boPin193Fault.AppScalingDivisor :=1;
boPin193Fault.AppScalingMultiplier :=1;
boPin193Fault.AppScalingOffset :=0;
boPin193Fault.AppUnit :="";
boPin193Fault.CanDefault :=0;
boPin193Fault.CanInit :=0;
boPin193Fault.CanMax :=1;
boPin193Fault.CanMin :=0;
boPin193Fault.CanUnit :="";
boPin193Fault.Description :="for the Neotec diag pages";
boPin193Fault.ErrorReaction := eErrorReaction.ERSIG_DFLT;
boPin193Fault.ReceiverAdress :=1;
boPin193Fault.ToolScalingDivisor :=1;
boPin193Fault.ToolScalingMultiplier :=1;
boPin193Fault.ToolScalingOffset :=0;
boPin193Fault.ToolUnit :="";

boPin169Fault.AppScalingDivisor :=1;
boPin169Fault.AppScalingMultiplier :=1;
boPin169Fault.AppScalingOffset :=0;
boPin169Fault.AppUnit :="";
boPin169Fault.CanDefault :=0;
boPin169Fault.CanInit :=0;
boPin169Fault.CanMax :=1;
boPin169Fault.CanMin :=0;
boPin169Fault.CanUnit :="";
boPin169Fault.Description :="for the Neotec diag pages";
boPin169Fault.ErrorReaction := eErrorReaction.ERSIG_DFLT;
boPin169Fault.ReceiverAdress :=1;
boPin169Fault.ToolScalingDivisor :=1;
boPin169Fault.ToolScalingMultiplier :=1;
boPin169Fault.ToolScalingOffset :=0;
boPin169Fault.ToolUnit :="";

boPin196Fault.AppScalingDivisor :=1;
boPin196Fault.AppScalingMultiplier :=1;
boPin196Fault.AppScalingOffset :=0;
boPin196Fault.AppUnit :="";
boPin196Fault.CanDefault :=0;
boPin196Fault.CanInit :=0;
boPin196Fault.CanMax :=1;
boPin196Fault.CanMin :=0;
boPin196Fault.CanUnit :="";
boPin196Fault.Description :="for the Neotec diag pages";
boPin196Fault.ErrorReaction := eErrorReaction.ERSIG_DFLT;
boPin196Fault.ReceiverAdress :=1;
boPin196Fault.ToolScalingDivisor :=1;
boPin196Fault.ToolScalingMultiplier :=1;
boPin196Fault.ToolScalingOffset :=0;
boPin196Fault.ToolUnit :="";

boPin172Fault.AppScalingDivisor :=1;
boPin172Fault.AppScalingMultiplier :=1;
boPin172Fault.AppScalingOffset :=0;
boPin172Fault.AppUnit :="";
boPin172Fault.CanDefault :=0;
boPin172Fault.CanInit :=0;
boPin172Fault.CanMax :=1;
boPin172Fault.CanMin :=0;
boPin172Fault.CanUnit :="";
boPin172Fault.Description :="for the Neotec diag pages";
boPin172Fault.ErrorReaction := eErrorReaction.ERSIG_DFLT;
boPin172Fault.ReceiverAdress :=1;
boPin172Fault.ToolScalingDivisor :=1;
boPin172Fault.ToolScalingMultiplier :=1;
boPin172Fault.ToolScalingOffset :=0;
boPin172Fault.ToolUnit :="";

boPin101Fault.AppScalingDivisor :=1;
boPin101Fault.AppScalingMultiplier :=1;
boPin101Fault.AppScalingOffset :=0;
boPin101Fault.AppUnit :="";
boPin101Fault.CanDefault :=0;
boPin101Fault.CanInit :=0;
boPin101Fault.CanMax :=1;
boPin101Fault.CanMin :=0;
boPin101Fault.CanUnit :="";
boPin101Fault.Description :="for the Neotec diag pages";
boPin101Fault.ErrorReaction := eErrorReaction.ERSIG_DFLT;
boPin101Fault.ReceiverAdress :=1;
boPin101Fault.ToolScalingDivisor :=1;
boPin101Fault.ToolScalingMultiplier :=1;
boPin101Fault.ToolScalingOffset :=0;
boPin101Fault.ToolUnit :="";

boPin125Fault.AppScalingDivisor :=1;
boPin125Fault.AppScalingMultiplier :=1;
boPin125Fault.AppScalingOffset :=0;
boPin125Fault.AppUnit :="";
boPin125Fault.CanDefault :=0;
boPin125Fault.CanInit :=0;
boPin125Fault.CanMax :=1;
boPin125Fault.CanMin :=0;
boPin125Fault.CanUnit :="";
boPin125Fault.Description :="for the Neotec diag pages";
boPin125Fault.ErrorReaction := eErrorReaction.ERSIG_DFLT;
boPin125Fault.ReceiverAdress :=1;
boPin125Fault.ToolScalingDivisor :=1;
boPin125Fault.ToolScalingMultiplier :=1;
boPin125Fault.ToolScalingOffset :=0;
boPin125Fault.ToolUnit :="";

boPin150Fault.AppScalingDivisor :=1;
boPin150Fault.AppScalingMultiplier :=1;
boPin150Fault.AppScalingOffset :=0;
boPin150Fault.AppUnit :="";
boPin150Fault.CanDefault :=0;
boPin150Fault.CanInit :=0;
boPin150Fault.CanMax :=1;
boPin150Fault.CanMin :=0;
boPin150Fault.CanUnit :="";
boPin150Fault.Description :="for the Neotec diag pages";
boPin150Fault.ErrorReaction := eErrorReaction.ERSIG_DFLT;
boPin150Fault.ReceiverAdress :=1;
boPin150Fault.ToolScalingDivisor :=1;
boPin150Fault.ToolScalingMultiplier :=1;
boPin150Fault.ToolScalingOffset :=0;
boPin150Fault.ToolUnit :="";

boPin174Fault.AppScalingDivisor :=1;
boPin174Fault.AppScalingMultiplier :=1;
boPin174Fault.AppScalingOffset :=0;
boPin174Fault.AppUnit :="";
boPin174Fault.CanDefault :=0;
boPin174Fault.CanInit :=0;
boPin174Fault.CanMax :=1;
boPin174Fault.CanMin :=0;
boPin174Fault.CanUnit :="";
boPin174Fault.Description :="for the Neotec diag pages";
boPin174Fault.ErrorReaction := eErrorReaction.ERSIG_DFLT;
boPin174Fault.ReceiverAdress :=1;
boPin174Fault.ToolScalingDivisor :=1;
boPin174Fault.ToolScalingMultiplier :=1;
boPin174Fault.ToolScalingOffset :=0;
boPin174Fault.ToolUnit :="";

boPin102Fault.AppScalingDivisor :=1;
boPin102Fault.AppScalingMultiplier :=1;
boPin102Fault.AppScalingOffset :=0;
boPin102Fault.AppUnit :="";
boPin102Fault.CanDefault :=0;
boPin102Fault.CanInit :=0;
boPin102Fault.CanMax :=1;
boPin102Fault.CanMin :=0;
boPin102Fault.CanUnit :="";
boPin102Fault.Description :="for the Neotec diag pages";
boPin102Fault.ErrorReaction := eErrorReaction.ERSIG_DFLT;
boPin102Fault.ReceiverAdress :=1;
boPin102Fault.ToolScalingDivisor :=1;
boPin102Fault.ToolScalingMultiplier :=1;
boPin102Fault.ToolScalingOffset :=0;
boPin102Fault.ToolUnit :="";

boPin126Fault.AppScalingDivisor :=1;
boPin126Fault.AppScalingMultiplier :=1;
boPin126Fault.AppScalingOffset :=0;
boPin126Fault.AppUnit :="";
boPin126Fault.CanDefault :=0;
boPin126Fault.CanInit :=0;
boPin126Fault.CanMax :=1;
boPin126Fault.CanMin :=0;
boPin126Fault.CanUnit :="";
boPin126Fault.Description :="for the Neotec diag pages";
boPin126Fault.ErrorReaction := eErrorReaction.ERSIG_DFLT;
boPin126Fault.ReceiverAdress :=1;
boPin126Fault.ToolScalingDivisor :=1;
boPin126Fault.ToolScalingMultiplier :=1;
boPin126Fault.ToolScalingOffset :=0;
boPin126Fault.ToolUnit :="";

boPin151Fault.AppScalingDivisor :=1;
boPin151Fault.AppScalingMultiplier :=1;
boPin151Fault.AppScalingOffset :=0;
boPin151Fault.AppUnit :="";
boPin151Fault.CanDefault :=0;
boPin151Fault.CanInit :=0;
boPin151Fault.CanMax :=1;
boPin151Fault.CanMin :=0;
boPin151Fault.CanUnit :="";
boPin151Fault.Description :="for the Neotec diag pages";
boPin151Fault.ErrorReaction := eErrorReaction.ERSIG_DFLT;
boPin151Fault.ReceiverAdress :=1;
boPin151Fault.ToolScalingDivisor :=1;
boPin151Fault.ToolScalingMultiplier :=1;
boPin151Fault.ToolScalingOffset :=0;
boPin151Fault.ToolUnit :="";

boPin175Fault.AppScalingDivisor :=1;
boPin175Fault.AppScalingMultiplier :=1;
boPin175Fault.AppScalingOffset :=0;
boPin175Fault.AppUnit :="";
boPin175Fault.CanDefault :=0;
boPin175Fault.CanInit :=0;
boPin175Fault.CanMax :=1;
boPin175Fault.CanMin :=0;
boPin175Fault.CanUnit :="";
boPin175Fault.Description :="for the Neotec diag pages";
boPin175Fault.ErrorReaction := eErrorReaction.ERSIG_DFLT;
boPin175Fault.ReceiverAdress :=1;
boPin175Fault.ToolScalingDivisor :=1;
boPin175Fault.ToolScalingMultiplier :=1;
boPin175Fault.ToolScalingOffset :=0;
boPin175Fault.ToolUnit :="";

boPin149Fault.AppScalingDivisor :=1;
boPin149Fault.AppScalingMultiplier :=1;
boPin149Fault.AppScalingOffset :=0;
boPin149Fault.AppUnit :="";
boPin149Fault.CanDefault :=0;
boPin149Fault.CanInit :=0;
boPin149Fault.CanMax :=1;
boPin149Fault.CanMin :=0;
boPin149Fault.CanUnit :="";
boPin149Fault.Description :="for the Neotec diag pages";
boPin149Fault.ErrorReaction := eErrorReaction.ERSIG_DFLT;
boPin149Fault.ReceiverAdress :=1;
boPin149Fault.ToolScalingDivisor :=1;
boPin149Fault.ToolScalingMultiplier :=1;
boPin149Fault.ToolScalingOffset :=0;
boPin149Fault.ToolUnit :="";

boPin173Fault.AppScalingDivisor :=1;
boPin173Fault.AppScalingMultiplier :=1;
boPin173Fault.AppScalingOffset :=0;
boPin173Fault.AppUnit :="";
boPin173Fault.CanDefault :=0;
boPin173Fault.CanInit :=0;
boPin173Fault.CanMax :=1;
boPin173Fault.CanMin :=0;
boPin173Fault.CanUnit :="";
boPin173Fault.Description :="for the Neotec diag pages";
boPin173Fault.ErrorReaction := eErrorReaction.ERSIG_DFLT;
boPin173Fault.ReceiverAdress :=1;
boPin173Fault.ToolScalingDivisor :=1;
boPin173Fault.ToolScalingMultiplier :=1;
boPin173Fault.ToolScalingOffset :=0;
boPin173Fault.ToolUnit :="";

boPin152Fault.AppScalingDivisor :=1;
boPin152Fault.AppScalingMultiplier :=1;
boPin152Fault.AppScalingOffset :=0;
boPin152Fault.AppUnit :="";
boPin152Fault.CanDefault :=0;
boPin152Fault.CanInit :=0;
boPin152Fault.CanMax :=1;
boPin152Fault.CanMin :=0;
boPin152Fault.CanUnit :="";
boPin152Fault.Description :="for the Neotec diag pages";
boPin152Fault.ErrorReaction := eErrorReaction.ERSIG_DFLT;
boPin152Fault.ReceiverAdress :=1;
boPin152Fault.ToolScalingDivisor :=1;
boPin152Fault.ToolScalingMultiplier :=1;
boPin152Fault.ToolScalingOffset :=0;
boPin152Fault.ToolUnit :="";

boPin176Fault.AppScalingDivisor :=1;
boPin176Fault.AppScalingMultiplier :=1;
boPin176Fault.AppScalingOffset :=0;
boPin176Fault.AppUnit :="";
boPin176Fault.CanDefault :=0;
boPin176Fault.CanInit :=0;
boPin176Fault.CanMax :=1;
boPin176Fault.CanMin :=0;
boPin176Fault.CanUnit :="";
boPin176Fault.Description :="for the Neotec diag pages";
boPin176Fault.ErrorReaction := eErrorReaction.ERSIG_DFLT;
boPin176Fault.ReceiverAdress :=1;
boPin176Fault.ToolScalingDivisor :=1;
boPin176Fault.ToolScalingMultiplier :=1;
boPin176Fault.ToolScalingOffset :=0;
boPin176Fault.ToolUnit :="";

boPin155Fault.AppScalingDivisor :=1;
boPin155Fault.AppScalingMultiplier :=1;
boPin155Fault.AppScalingOffset :=0;
boPin155Fault.AppUnit :="";
boPin155Fault.CanDefault :=0;
boPin155Fault.CanInit :=0;
boPin155Fault.CanMax :=1;
boPin155Fault.CanMin :=0;
boPin155Fault.CanUnit :="";
boPin155Fault.Description :="for the Neotec diag pages";
boPin155Fault.ErrorReaction := eErrorReaction.ERSIG_DFLT;
boPin155Fault.ReceiverAdress :=1;
boPin155Fault.ToolScalingDivisor :=1;
boPin155Fault.ToolScalingMultiplier :=1;
boPin155Fault.ToolScalingOffset :=0;
boPin155Fault.ToolUnit :="";

boPin179Fault.AppScalingDivisor :=1;
boPin179Fault.AppScalingMultiplier :=1;
boPin179Fault.AppScalingOffset :=0;
boPin179Fault.AppUnit :="";
boPin179Fault.CanDefault :=0;
boPin179Fault.CanInit :=0;
boPin179Fault.CanMax :=1;
boPin179Fault.CanMin :=0;
boPin179Fault.CanUnit :="";
boPin179Fault.Description :="for the Neotec diag pages";
boPin179Fault.ErrorReaction := eErrorReaction.ERSIG_DFLT;
boPin179Fault.ReceiverAdress :=1;
boPin179Fault.ToolScalingDivisor :=1;
boPin179Fault.ToolScalingMultiplier :=1;
boPin179Fault.ToolScalingOffset :=0;
boPin179Fault.ToolUnit :="";

boPin158Fault.AppScalingDivisor :=1;
boPin158Fault.AppScalingMultiplier :=1;
boPin158Fault.AppScalingOffset :=0;
boPin158Fault.AppUnit :="";
boPin158Fault.CanDefault :=0;
boPin158Fault.CanInit :=0;
boPin158Fault.CanMax :=1;
boPin158Fault.CanMin :=0;
boPin158Fault.CanUnit :="";
boPin158Fault.Description :="for the Neotec diag pages";
boPin158Fault.ErrorReaction := eErrorReaction.ERSIG_DFLT;
boPin158Fault.ReceiverAdress :=1;
boPin158Fault.ToolScalingDivisor :=1;
boPin158Fault.ToolScalingMultiplier :=1;
boPin158Fault.ToolScalingOffset :=0;
boPin158Fault.ToolUnit :="";

boPin182Fault.AppScalingDivisor :=1;
boPin182Fault.AppScalingMultiplier :=1;
boPin182Fault.AppScalingOffset :=0;
boPin182Fault.AppUnit :="";
boPin182Fault.CanDefault :=0;
boPin182Fault.CanInit :=0;
boPin182Fault.CanMax :=1;
boPin182Fault.CanMin :=0;
boPin182Fault.CanUnit :="";
boPin182Fault.Description :="for the Neotec diag pages";
boPin182Fault.ErrorReaction := eErrorReaction.ERSIG_DFLT;
boPin182Fault.ReceiverAdress :=1;
boPin182Fault.ToolScalingDivisor :=1;
boPin182Fault.ToolScalingMultiplier :=1;
boPin182Fault.ToolScalingOffset :=0;
boPin182Fault.ToolUnit :="";

boPin251Fault.AppScalingDivisor :=1;
boPin251Fault.AppScalingMultiplier :=1;
boPin251Fault.AppScalingOffset :=0;
boPin251Fault.AppUnit :="";
boPin251Fault.CanDefault :=0;
boPin251Fault.CanInit :=0;
boPin251Fault.CanMax :=1;
boPin251Fault.CanMin :=0;
boPin251Fault.CanUnit :="";
boPin251Fault.Description :="for the Neotec diag pages";
boPin251Fault.ErrorReaction := eErrorReaction.ERSIG_DFLT;
boPin251Fault.ReceiverAdress :=1;
boPin251Fault.ToolScalingDivisor :=1;
boPin251Fault.ToolScalingMultiplier :=1;
boPin251Fault.ToolScalingOffset :=0;
boPin251Fault.ToolUnit :="";

boPin238Fault.AppScalingDivisor :=1;
boPin238Fault.AppScalingMultiplier :=1;
boPin238Fault.AppScalingOffset :=0;
boPin238Fault.AppUnit :="";
boPin238Fault.CanDefault :=0;
boPin238Fault.CanInit :=0;
boPin238Fault.CanMax :=1;
boPin238Fault.CanMin :=0;
boPin238Fault.CanUnit :="";
boPin238Fault.Description :="for the Neotec diag pages";
boPin238Fault.ErrorReaction := eErrorReaction.ERSIG_DFLT;
boPin238Fault.ReceiverAdress :=1;
boPin238Fault.ToolScalingDivisor :=1;
boPin238Fault.ToolScalingMultiplier :=1;
boPin238Fault.ToolScalingOffset :=0;
boPin238Fault.ToolUnit :="";

boPin252Fault.AppScalingDivisor :=1;
boPin252Fault.AppScalingMultiplier :=1;
boPin252Fault.AppScalingOffset :=0;
boPin252Fault.AppUnit :="";
boPin252Fault.CanDefault :=0;
boPin252Fault.CanInit :=0;
boPin252Fault.CanMax :=1;
boPin252Fault.CanMin :=0;
boPin252Fault.CanUnit :="";
boPin252Fault.Description :="for the Neotec diag pages";
boPin252Fault.ErrorReaction := eErrorReaction.ERSIG_DFLT;
boPin252Fault.ReceiverAdress :=1;
boPin252Fault.ToolScalingDivisor :=1;
boPin252Fault.ToolScalingMultiplier :=1;
boPin252Fault.ToolScalingOffset :=0;
boPin252Fault.ToolUnit :="";

boPin239Fault.AppScalingDivisor :=1;
boPin239Fault.AppScalingMultiplier :=1;
boPin239Fault.AppScalingOffset :=0;
boPin239Fault.AppUnit :="";
boPin239Fault.CanDefault :=0;
boPin239Fault.CanInit :=0;
boPin239Fault.CanMax :=1;
boPin239Fault.CanMin :=0;
boPin239Fault.CanUnit :="";
boPin239Fault.Description :="for the Neotec diag pages";
boPin239Fault.ErrorReaction := eErrorReaction.ERSIG_DFLT;
boPin239Fault.ReceiverAdress :=1;
boPin239Fault.ToolScalingDivisor :=1;
boPin239Fault.ToolScalingMultiplier :=1;
boPin239Fault.ToolScalingOffset :=0;
boPin239Fault.ToolUnit :="";

boPin253Fault.AppScalingDivisor :=1;
boPin253Fault.AppScalingMultiplier :=1;
boPin253Fault.AppScalingOffset :=0;
boPin253Fault.AppUnit :="";
boPin253Fault.CanDefault :=0;
boPin253Fault.CanInit :=0;
boPin253Fault.CanMax :=1;
boPin253Fault.CanMin :=0;
boPin253Fault.CanUnit :="";
boPin253Fault.Description :="for the Neotec diag pages";
boPin253Fault.ErrorReaction := eErrorReaction.ERSIG_DFLT;
boPin253Fault.ReceiverAdress :=1;
boPin253Fault.ToolScalingDivisor :=1;
boPin253Fault.ToolScalingMultiplier :=1;
boPin253Fault.ToolScalingOffset :=0;
boPin253Fault.ToolUnit :="";

boPin240Fault.AppScalingDivisor :=1;
boPin240Fault.AppScalingMultiplier :=1;
boPin240Fault.AppScalingOffset :=0;
boPin240Fault.AppUnit :="";
boPin240Fault.CanDefault :=0;
boPin240Fault.CanInit :=0;
boPin240Fault.CanMax :=1;
boPin240Fault.CanMin :=0;
boPin240Fault.CanUnit :="";
boPin240Fault.Description :="for the Neotec diag pages";
boPin240Fault.ErrorReaction := eErrorReaction.ERSIG_DFLT;
boPin240Fault.ReceiverAdress :=1;
boPin240Fault.ToolScalingDivisor :=1;
boPin240Fault.ToolScalingMultiplier :=1;
boPin240Fault.ToolScalingOffset :=0;
boPin240Fault.ToolUnit :="";

boPin254Fault.AppScalingDivisor :=1;
boPin254Fault.AppScalingMultiplier :=1;
boPin254Fault.AppScalingOffset :=0;
boPin254Fault.AppUnit :="";
boPin254Fault.CanDefault :=0;
boPin254Fault.CanInit :=0;
boPin254Fault.CanMax :=1;
boPin254Fault.CanMin :=0;
boPin254Fault.CanUnit :="";
boPin254Fault.Description :="for the Neotec diag pages";
boPin254Fault.ErrorReaction := eErrorReaction.ERSIG_DFLT;
boPin254Fault.ReceiverAdress :=1;
boPin254Fault.ToolScalingDivisor :=1;
boPin254Fault.ToolScalingMultiplier :=1;
boPin254Fault.ToolScalingOffset :=0;
boPin254Fault.ToolUnit :="";

boPin241Fault.AppScalingDivisor :=1;
boPin241Fault.AppScalingMultiplier :=1;
boPin241Fault.AppScalingOffset :=0;
boPin241Fault.AppUnit :="";
boPin241Fault.CanDefault :=0;
boPin241Fault.CanInit :=0;
boPin241Fault.CanMax :=1;
boPin241Fault.CanMin :=0;
boPin241Fault.CanUnit :="";
boPin241Fault.Description :="for the Neotec diag pages";
boPin241Fault.ErrorReaction := eErrorReaction.ERSIG_DFLT;
boPin241Fault.ReceiverAdress :=1;
boPin241Fault.ToolScalingDivisor :=1;
boPin241Fault.ToolScalingMultiplier :=1;
boPin241Fault.ToolScalingOffset :=0;
boPin241Fault.ToolUnit :="";

boPin161Fault.AppScalingDivisor :=1;
boPin161Fault.AppScalingMultiplier :=1;
boPin161Fault.AppScalingOffset :=0;
boPin161Fault.AppUnit :="";
boPin161Fault.CanDefault :=0;
boPin161Fault.CanInit :=0;
boPin161Fault.CanMax :=1;
boPin161Fault.CanMin :=0;
boPin161Fault.CanUnit :="";
boPin161Fault.Description :="for the Neotec diag pages";
boPin161Fault.ErrorReaction := eErrorReaction.ERSIG_DFLT;
boPin161Fault.ReceiverAdress :=1;
boPin161Fault.ToolScalingDivisor :=1;
boPin161Fault.ToolScalingMultiplier :=1;
boPin161Fault.ToolScalingOffset :=0;
boPin161Fault.ToolUnit :="";

boPin185Fault.AppScalingDivisor :=1;
boPin185Fault.AppScalingMultiplier :=1;
boPin185Fault.AppScalingOffset :=0;
boPin185Fault.AppUnit :="";
boPin185Fault.CanDefault :=0;
boPin185Fault.CanInit :=0;
boPin185Fault.CanMax :=1;
boPin185Fault.CanMin :=0;
boPin185Fault.CanUnit :="";
boPin185Fault.Description :="for the Neotec diag pages";
boPin185Fault.ErrorReaction := eErrorReaction.ERSIG_DFLT;
boPin185Fault.ReceiverAdress :=1;
boPin185Fault.ToolScalingDivisor :=1;
boPin185Fault.ToolScalingMultiplier :=1;
boPin185Fault.ToolScalingOffset :=0;
boPin185Fault.ToolUnit :="";

boPin188Fault.AppScalingDivisor :=1;
boPin188Fault.AppScalingMultiplier :=1;
boPin188Fault.AppScalingOffset :=0;
boPin188Fault.AppUnit :="";
boPin188Fault.CanDefault :=0;
boPin188Fault.CanInit :=0;
boPin188Fault.CanMax :=1;
boPin188Fault.CanMin :=0;
boPin188Fault.CanUnit :="";
boPin188Fault.Description :="for the Neotec diag pages";
boPin188Fault.ErrorReaction := eErrorReaction.ERSIG_DFLT;
boPin188Fault.ReceiverAdress :=1;
boPin188Fault.ToolScalingDivisor :=1;
boPin188Fault.ToolScalingMultiplier :=1;
boPin188Fault.ToolScalingOffset :=0;
boPin188Fault.ToolUnit :="";

boPin164Fault.AppScalingDivisor :=1;
boPin164Fault.AppScalingMultiplier :=1;
boPin164Fault.AppScalingOffset :=0;
boPin164Fault.AppUnit :="";
boPin164Fault.CanDefault :=0;
boPin164Fault.CanInit :=0;
boPin164Fault.CanMax :=1;
boPin164Fault.CanMin :=0;
boPin164Fault.CanUnit :="";
boPin164Fault.Description :="for the Neotec diag pages";
boPin164Fault.ErrorReaction := eErrorReaction.ERSIG_DFLT;
boPin164Fault.ReceiverAdress :=1;
boPin164Fault.ToolScalingDivisor :=1;
boPin164Fault.ToolScalingMultiplier :=1;
boPin164Fault.ToolScalingOffset :=0;
boPin164Fault.ToolUnit :="";

boPin191Fault.AppScalingDivisor :=1;
boPin191Fault.AppScalingMultiplier :=1;
boPin191Fault.AppScalingOffset :=0;
boPin191Fault.AppUnit :="";
boPin191Fault.CanDefault :=0;
boPin191Fault.CanInit :=0;
boPin191Fault.CanMax :=1;
boPin191Fault.CanMin :=0;
boPin191Fault.CanUnit :="";
boPin191Fault.Description :="for the Neotec diag pages";
boPin191Fault.ErrorReaction := eErrorReaction.ERSIG_DFLT;
boPin191Fault.ReceiverAdress :=1;
boPin191Fault.ToolScalingDivisor :=1;
boPin191Fault.ToolScalingMultiplier :=1;
boPin191Fault.ToolScalingOffset :=0;
boPin191Fault.ToolUnit :="";

boPin167Fault.AppScalingDivisor :=1;
boPin167Fault.AppScalingMultiplier :=1;
boPin167Fault.AppScalingOffset :=0;
boPin167Fault.AppUnit :="";
boPin167Fault.CanDefault :=0;
boPin167Fault.CanInit :=0;
boPin167Fault.CanMax :=1;
boPin167Fault.CanMin :=0;
boPin167Fault.CanUnit :="";
boPin167Fault.Description :="for the Neotec diag pages";
boPin167Fault.ErrorReaction := eErrorReaction.ERSIG_DFLT;
boPin167Fault.ReceiverAdress :=1;
boPin167Fault.ToolScalingDivisor :=1;
boPin167Fault.ToolScalingMultiplier :=1;
boPin167Fault.ToolScalingOffset :=0;
boPin167Fault.ToolUnit :="";

boPin194Fault.AppScalingDivisor :=1;
boPin194Fault.AppScalingMultiplier :=1;
boPin194Fault.AppScalingOffset :=0;
boPin194Fault.AppUnit :="";
boPin194Fault.CanDefault :=0;
boPin194Fault.CanInit :=0;
boPin194Fault.CanMax :=1;
boPin194Fault.CanMin :=0;
boPin194Fault.CanUnit :="";
boPin194Fault.Description :="for the Neotec diag pages";
boPin194Fault.ErrorReaction := eErrorReaction.ERSIG_DFLT;
boPin194Fault.ReceiverAdress :=1;
boPin194Fault.ToolScalingDivisor :=1;
boPin194Fault.ToolScalingMultiplier :=1;
boPin194Fault.ToolScalingOffset :=0;
boPin194Fault.ToolUnit :="";

boPin170Fault.AppScalingDivisor :=1;
boPin170Fault.AppScalingMultiplier :=1;
boPin170Fault.AppScalingOffset :=0;
boPin170Fault.AppUnit :="";
boPin170Fault.CanDefault :=0;
boPin170Fault.CanInit :=0;
boPin170Fault.CanMax :=1;
boPin170Fault.CanMin :=0;
boPin170Fault.CanUnit :="";
boPin170Fault.Description :="for the Neotec diag pages";
boPin170Fault.ErrorReaction := eErrorReaction.ERSIG_DFLT;
boPin170Fault.ReceiverAdress :=1;
boPin170Fault.ToolScalingDivisor :=1;
boPin170Fault.ToolScalingMultiplier :=1;
boPin170Fault.ToolScalingOffset :=0;
boPin170Fault.ToolUnit :="";


                
END_METHOD
END_FUNCTION_BLOCK

FUNCTION_BLOCK Msg7C0SendToEvision7MessageClass EXTENDS CanReceiveMessageClass
  VAR_INPUT
    boPin107 : BoolCanSignalClass;
    boPin131 : BoolCanSignalClass;
    boPin108 : BoolCanSignalClass;
    boPin132 : BoolCanSignalClass;
    boPin109 : BoolCanSignalClass;
    boPin133 : BoolCanSignalClass;
    boPin110 : BoolCanSignalClass;
    boPin134 : BoolCanSignalClass;
    boPin111 : BoolCanSignalClass;
    boPin135 : BoolCanSignalClass;
    boPin112 : BoolCanSignalClass;
    boPin136 : BoolCanSignalClass;
    boPin113 : BoolCanSignalClass;
    boPin137 : BoolCanSignalClass;
    boPin114 : BoolCanSignalClass;
    boPin138 : BoolCanSignalClass;
    boPin140 : BoolCanSignalClass;
    boPin117 : BoolCanSignalClass;
    boPin141 : BoolCanSignalClass;
    boPin122 : BoolCanSignalClass;
    boPin146 : BoolCanSignalClass;
    boPin123 : BoolCanSignalClass;
    boPin187 : BoolCanSignalClass;
    boPin124 : BoolCanSignalClass;
    boPin148 : BoolCanSignalClass;
    boPin153 : BoolCanSignalClass;
    boPin177 : BoolCanSignalClass;
    boPin156 : BoolCanSignalClass;
    boPin159 : BoolCanSignalClass;
    boPin186 : BoolCanSignalClass;
    boPin162 : BoolCanSignalClass;
    boPin189 : BoolCanSignalClass;
    boPin165 : BoolCanSignalClass;
    boPin195 : BoolCanSignalClass;
    boPin171 : BoolCanSignalClass;
    boPin154 : BoolCanSignalClass;
    boPin160 : BoolCanSignalClass;
    boPin184 : BoolCanSignalClass;
    boPin163 : BoolCanSignalClass;
    boPin190 : BoolCanSignalClass;
    boPin166 : BoolCanSignalClass;
    boPin193 : BoolCanSignalClass;
    boPin169 : BoolCanSignalClass;
    boPin196 : BoolCanSignalClass;
    boPin172 : BoolCanSignalClass;
    boPin149 : BoolCanSignalClass;
    boPin173 : BoolCanSignalClass;
    boPin152 : BoolCanSignalClass;
    boPin176 : BoolCanSignalClass;
    boPin155 : BoolCanSignalClass;
    boPin179 : BoolCanSignalClass;
    boPin158 : BoolCanSignalClass;
    boPin182 : BoolCanSignalClass;
    boPin252 : BoolCanSignalClass;
    boPin239 : BoolCanSignalClass;
    boPin188 : BoolCanSignalClass;
    boPin164 : BoolCanSignalClass;
    boPin191 : BoolCanSignalClass;
    boPin167 : BoolCanSignalClass;
    boPin194 : BoolCanSignalClass;
    boPin170 : BoolCanSignalClass;
    boPin192 : BoolCanSignalClass;
    boPin168 : BoolCanSignalClass;
    Counter : UInt32CanSignalClass;
  END_VAR

            
          

METHOD SetData
  VAR_INPUT
    CanMsgPointer : POINTER TO CanMessageClass;
  END_VAR
                  IF IsValidPointer(canMsgPointer,'SetData') THEN
	SUPER^.SetData(CanMsgPointer);
	//Set the new data
	boPin107.Value := canMsgPointer^.GetBoolOnBit(0);
	boPin131.Value := canMsgPointer^.GetBoolOnBit(1);
	boPin108.Value := canMsgPointer^.GetBoolOnBit(2);
	boPin132.Value := canMsgPointer^.GetBoolOnBit(3);
	boPin109.Value := canMsgPointer^.GetBoolOnBit(4);
	boPin133.Value := canMsgPointer^.GetBoolOnBit(5);
	boPin110.Value := canMsgPointer^.GetBoolOnBit(6);
	boPin134.Value := canMsgPointer^.GetBoolOnBit(7);
	boPin111.Value := canMsgPointer^.GetBoolOnBit(8);
	boPin135.Value := canMsgPointer^.GetBoolOnBit(9);
	boPin112.Value := canMsgPointer^.GetBoolOnBit(10);
	boPin136.Value := canMsgPointer^.GetBoolOnBit(11);
	boPin113.Value := canMsgPointer^.GetBoolOnBit(12);
	boPin137.Value := canMsgPointer^.GetBoolOnBit(13);
	boPin114.Value := canMsgPointer^.GetBoolOnBit(14);
	boPin138.Value := canMsgPointer^.GetBoolOnBit(15);
	boPin140.Value := canMsgPointer^.GetBoolOnBit(16);
	boPin117.Value := canMsgPointer^.GetBoolOnBit(17);
	boPin141.Value := canMsgPointer^.GetBoolOnBit(18);
	boPin122.Value := canMsgPointer^.GetBoolOnBit(19);
	boPin146.Value := canMsgPointer^.GetBoolOnBit(20);
	boPin123.Value := canMsgPointer^.GetBoolOnBit(21);
	boPin187.Value := canMsgPointer^.GetBoolOnBit(22);
	boPin124.Value := canMsgPointer^.GetBoolOnBit(23);
	boPin148.Value := canMsgPointer^.GetBoolOnBit(24);
	boPin153.Value := canMsgPointer^.GetBoolOnBit(25);
	boPin177.Value := canMsgPointer^.GetBoolOnBit(26);
	boPin156.Value := canMsgPointer^.GetBoolOnBit(27);
	boPin159.Value := canMsgPointer^.GetBoolOnBit(28);
	boPin186.Value := canMsgPointer^.GetBoolOnBit(29);
	boPin162.Value := canMsgPointer^.GetBoolOnBit(30);
	boPin189.Value := canMsgPointer^.GetBoolOnBit(31);
	boPin165.Value := canMsgPointer^.GetBoolOnBit(32);
	boPin195.Value := canMsgPointer^.GetBoolOnBit(33);
	boPin171.Value := canMsgPointer^.GetBoolOnBit(34);
	boPin154.Value := canMsgPointer^.GetBoolOnBit(35);
	boPin160.Value := canMsgPointer^.GetBoolOnBit(36);
	boPin184.Value := canMsgPointer^.GetBoolOnBit(37);
	boPin163.Value := canMsgPointer^.GetBoolOnBit(38);
	boPin190.Value := canMsgPointer^.GetBoolOnBit(39);
	boPin166.Value := canMsgPointer^.GetBoolOnBit(40);
	boPin193.Value := canMsgPointer^.GetBoolOnBit(41);
	boPin169.Value := canMsgPointer^.GetBoolOnBit(42);
	boPin196.Value := canMsgPointer^.GetBoolOnBit(43);
	boPin172.Value := canMsgPointer^.GetBoolOnBit(44);
	boPin149.Value := canMsgPointer^.GetBoolOnBit(45);
	boPin173.Value := canMsgPointer^.GetBoolOnBit(46);
	boPin152.Value := canMsgPointer^.GetBoolOnBit(47);
	boPin176.Value := canMsgPointer^.GetBoolOnBit(48);
	boPin155.Value := canMsgPointer^.GetBoolOnBit(49);
	boPin179.Value := canMsgPointer^.GetBoolOnBit(50);
	boPin158.Value := canMsgPointer^.GetBoolOnBit(51);
	boPin182.Value := canMsgPointer^.GetBoolOnBit(52);
	boPin252.Value := canMsgPointer^.GetBoolOnBit(53);
	boPin239.Value := canMsgPointer^.GetBoolOnBit(54);
	boPin188.Value := canMsgPointer^.GetBoolOnBit(55);
	boPin164.Value := canMsgPointer^.GetBoolOnBit(56);
	boPin191.Value := canMsgPointer^.GetBoolOnBit(57);
	boPin167.Value := canMsgPointer^.GetBoolOnBit(58);
	boPin194.Value := canMsgPointer^.GetBoolOnBit(59);
	boPin170.Value := canMsgPointer^.GetBoolOnBit(60);
	boPin192.Value := canMsgPointer^.GetBoolOnBit(61);
	boPin168.Value := canMsgPointer^.GetBoolOnBit(62);
	//And increase the counter
	Counter.Value := CanMsgPointer^.Counter.Value;
END_IF

                
END_METHOD

PROPERTY boPin107RawValue : BOOL
GET
                    boPin107RawValue := boPin107.Value;

                  
END_GET
END_PROPERTY

PROPERTY boPin131RawValue : BOOL
GET
                    boPin131RawValue := boPin131.Value;

                  
END_GET
END_PROPERTY

PROPERTY boPin108RawValue : BOOL
GET
                    boPin108RawValue := boPin108.Value;

                  
END_GET
END_PROPERTY

PROPERTY boPin132RawValue : BOOL
GET
                    boPin132RawValue := boPin132.Value;

                  
END_GET
END_PROPERTY

PROPERTY boPin109RawValue : BOOL
GET
                    boPin109RawValue := boPin109.Value;

                  
END_GET
END_PROPERTY

PROPERTY boPin133RawValue : BOOL
GET
                    boPin133RawValue := boPin133.Value;

                  
END_GET
END_PROPERTY

PROPERTY boPin110RawValue : BOOL
GET
                    boPin110RawValue := boPin110.Value;

                  
END_GET
END_PROPERTY

PROPERTY boPin134RawValue : BOOL
GET
                    boPin134RawValue := boPin134.Value;

                  
END_GET
END_PROPERTY

PROPERTY boPin111RawValue : BOOL
GET
                    boPin111RawValue := boPin111.Value;

                  
END_GET
END_PROPERTY

PROPERTY boPin135RawValue : BOOL
GET
                    boPin135RawValue := boPin135.Value;

                  
END_GET
END_PROPERTY

PROPERTY boPin112RawValue : BOOL
GET
                    boPin112RawValue := boPin112.Value;

                  
END_GET
END_PROPERTY

PROPERTY boPin136RawValue : BOOL
GET
                    boPin136RawValue := boPin136.Value;

                  
END_GET
END_PROPERTY

PROPERTY boPin113RawValue : BOOL
GET
                    boPin113RawValue := boPin113.Value;

                  
END_GET
END_PROPERTY

PROPERTY boPin137RawValue : BOOL
GET
                    boPin137RawValue := boPin137.Value;

                  
END_GET
END_PROPERTY

PROPERTY boPin114RawValue : BOOL
GET
                    boPin114RawValue := boPin114.Value;

                  
END_GET
END_PROPERTY

PROPERTY boPin138RawValue : BOOL
GET
                    boPin138RawValue := boPin138.Value;

                  
END_GET
END_PROPERTY

PROPERTY boPin140RawValue : BOOL
GET
                    boPin140RawValue := boPin140.Value;

                  
END_GET
END_PROPERTY

PROPERTY boPin117RawValue : BOOL
GET
                    boPin117RawValue := boPin117.Value;

                  
END_GET
END_PROPERTY

PROPERTY boPin141RawValue : BOOL
GET
                    boPin141RawValue := boPin141.Value;

                  
END_GET
END_PROPERTY

PROPERTY boPin122RawValue : BOOL
GET
                    boPin122RawValue := boPin122.Value;

                  
END_GET
END_PROPERTY

PROPERTY boPin146RawValue : BOOL
GET
                    boPin146RawValue := boPin146.Value;

                  
END_GET
END_PROPERTY

PROPERTY boPin123RawValue : BOOL
GET
                    boPin123RawValue := boPin123.Value;

                  
END_GET
END_PROPERTY

PROPERTY boPin187RawValue : BOOL
GET
                    boPin187RawValue := boPin187.Value;

                  
END_GET
END_PROPERTY

PROPERTY boPin124RawValue : BOOL
GET
                    boPin124RawValue := boPin124.Value;

                  
END_GET
END_PROPERTY

PROPERTY boPin148RawValue : BOOL
GET
                    boPin148RawValue := boPin148.Value;

                  
END_GET
END_PROPERTY

PROPERTY boPin153RawValue : BOOL
GET
                    boPin153RawValue := boPin153.Value;

                  
END_GET
END_PROPERTY

PROPERTY boPin177RawValue : BOOL
GET
                    boPin177RawValue := boPin177.Value;

                  
END_GET
END_PROPERTY

PROPERTY boPin156RawValue : BOOL
GET
                    boPin156RawValue := boPin156.Value;

                  
END_GET
END_PROPERTY

PROPERTY boPin159RawValue : BOOL
GET
                    boPin159RawValue := boPin159.Value;

                  
END_GET
END_PROPERTY

PROPERTY boPin186RawValue : BOOL
GET
                    boPin186RawValue := boPin186.Value;

                  
END_GET
END_PROPERTY

PROPERTY boPin162RawValue : BOOL
GET
                    boPin162RawValue := boPin162.Value;

                  
END_GET
END_PROPERTY

PROPERTY boPin189RawValue : BOOL
GET
                    boPin189RawValue := boPin189.Value;

                  
END_GET
END_PROPERTY

PROPERTY boPin165RawValue : BOOL
GET
                    boPin165RawValue := boPin165.Value;

                  
END_GET
END_PROPERTY

PROPERTY boPin195RawValue : BOOL
GET
                    boPin195RawValue := boPin195.Value;

                  
END_GET
END_PROPERTY

PROPERTY boPin171RawValue : BOOL
GET
                    boPin171RawValue := boPin171.Value;

                  
END_GET
END_PROPERTY

PROPERTY boPin154RawValue : BOOL
GET
                    boPin154RawValue := boPin154.Value;

                  
END_GET
END_PROPERTY

PROPERTY boPin160RawValue : BOOL
GET
                    boPin160RawValue := boPin160.Value;

                  
END_GET
END_PROPERTY

PROPERTY boPin184RawValue : BOOL
GET
                    boPin184RawValue := boPin184.Value;

                  
END_GET
END_PROPERTY

PROPERTY boPin163RawValue : BOOL
GET
                    boPin163RawValue := boPin163.Value;

                  
END_GET
END_PROPERTY

PROPERTY boPin190RawValue : BOOL
GET
                    boPin190RawValue := boPin190.Value;

                  
END_GET
END_PROPERTY

PROPERTY boPin166RawValue : BOOL
GET
                    boPin166RawValue := boPin166.Value;

                  
END_GET
END_PROPERTY

PROPERTY boPin193RawValue : BOOL
GET
                    boPin193RawValue := boPin193.Value;

                  
END_GET
END_PROPERTY

PROPERTY boPin169RawValue : BOOL
GET
                    boPin169RawValue := boPin169.Value;

                  
END_GET
END_PROPERTY

PROPERTY boPin196RawValue : BOOL
GET
                    boPin196RawValue := boPin196.Value;

                  
END_GET
END_PROPERTY

PROPERTY boPin172RawValue : BOOL
GET
                    boPin172RawValue := boPin172.Value;

                  
END_GET
END_PROPERTY

PROPERTY boPin149RawValue : BOOL
GET
                    boPin149RawValue := boPin149.Value;

                  
END_GET
END_PROPERTY

PROPERTY boPin173RawValue : BOOL
GET
                    boPin173RawValue := boPin173.Value;

                  
END_GET
END_PROPERTY

PROPERTY boPin152RawValue : BOOL
GET
                    boPin152RawValue := boPin152.Value;

                  
END_GET
END_PROPERTY

PROPERTY boPin176RawValue : BOOL
GET
                    boPin176RawValue := boPin176.Value;

                  
END_GET
END_PROPERTY

PROPERTY boPin155RawValue : BOOL
GET
                    boPin155RawValue := boPin155.Value;

                  
END_GET
END_PROPERTY

PROPERTY boPin179RawValue : BOOL
GET
                    boPin179RawValue := boPin179.Value;

                  
END_GET
END_PROPERTY

PROPERTY boPin158RawValue : BOOL
GET
                    boPin158RawValue := boPin158.Value;

                  
END_GET
END_PROPERTY

PROPERTY boPin182RawValue : BOOL
GET
                    boPin182RawValue := boPin182.Value;

                  
END_GET
END_PROPERTY

PROPERTY boPin252RawValue : BOOL
GET
                    boPin252RawValue := boPin252.Value;

                  
END_GET
END_PROPERTY

PROPERTY boPin239RawValue : BOOL
GET
                    boPin239RawValue := boPin239.Value;

                  
END_GET
END_PROPERTY

PROPERTY boPin188RawValue : BOOL
GET
                    boPin188RawValue := boPin188.Value;

                  
END_GET
END_PROPERTY

PROPERTY boPin164RawValue : BOOL
GET
                    boPin164RawValue := boPin164.Value;

                  
END_GET
END_PROPERTY

PROPERTY boPin191RawValue : BOOL
GET
                    boPin191RawValue := boPin191.Value;

                  
END_GET
END_PROPERTY

PROPERTY boPin167RawValue : BOOL
GET
                    boPin167RawValue := boPin167.Value;

                  
END_GET
END_PROPERTY

PROPERTY boPin194RawValue : BOOL
GET
                    boPin194RawValue := boPin194.Value;

                  
END_GET
END_PROPERTY

PROPERTY boPin170RawValue : BOOL
GET
                    boPin170RawValue := boPin170.Value;

                  
END_GET
END_PROPERTY

PROPERTY boPin192RawValue : BOOL
GET
                    boPin192RawValue := boPin192.Value;

                  
END_GET
END_PROPERTY

PROPERTY boPin168RawValue : BOOL
GET
                    boPin168RawValue := boPin168.Value;

                  
END_GET
END_PROPERTY

PROPERTY boPin107ToolValue : BOOL
GET
                    boPin107ToolValue := boPin107.Value;

                  
END_GET
END_PROPERTY

PROPERTY boPin131ToolValue : BOOL
GET
                    boPin131ToolValue := boPin131.Value;

                  
END_GET
END_PROPERTY

PROPERTY boPin108ToolValue : BOOL
GET
                    boPin108ToolValue := boPin108.Value;

                  
END_GET
END_PROPERTY

PROPERTY boPin132ToolValue : BOOL
GET
                    boPin132ToolValue := boPin132.Value;

                  
END_GET
END_PROPERTY

PROPERTY boPin109ToolValue : BOOL
GET
                    boPin109ToolValue := boPin109.Value;

                  
END_GET
END_PROPERTY

PROPERTY boPin133ToolValue : BOOL
GET
                    boPin133ToolValue := boPin133.Value;

                  
END_GET
END_PROPERTY

PROPERTY boPin110ToolValue : BOOL
GET
                    boPin110ToolValue := boPin110.Value;

                  
END_GET
END_PROPERTY

PROPERTY boPin134ToolValue : BOOL
GET
                    boPin134ToolValue := boPin134.Value;

                  
END_GET
END_PROPERTY

PROPERTY boPin111ToolValue : BOOL
GET
                    boPin111ToolValue := boPin111.Value;

                  
END_GET
END_PROPERTY

PROPERTY boPin135ToolValue : BOOL
GET
                    boPin135ToolValue := boPin135.Value;

                  
END_GET
END_PROPERTY

PROPERTY boPin112ToolValue : BOOL
GET
                    boPin112ToolValue := boPin112.Value;

                  
END_GET
END_PROPERTY

PROPERTY boPin136ToolValue : BOOL
GET
                    boPin136ToolValue := boPin136.Value;

                  
END_GET
END_PROPERTY

PROPERTY boPin113ToolValue : BOOL
GET
                    boPin113ToolValue := boPin113.Value;

                  
END_GET
END_PROPERTY

PROPERTY boPin137ToolValue : BOOL
GET
                    boPin137ToolValue := boPin137.Value;

                  
END_GET
END_PROPERTY

PROPERTY boPin114ToolValue : BOOL
GET
                    boPin114ToolValue := boPin114.Value;

                  
END_GET
END_PROPERTY

PROPERTY boPin138ToolValue : BOOL
GET
                    boPin138ToolValue := boPin138.Value;

                  
END_GET
END_PROPERTY

PROPERTY boPin140ToolValue : BOOL
GET
                    boPin140ToolValue := boPin140.Value;

                  
END_GET
END_PROPERTY

PROPERTY boPin117ToolValue : BOOL
GET
                    boPin117ToolValue := boPin117.Value;

                  
END_GET
END_PROPERTY

PROPERTY boPin141ToolValue : BOOL
GET
                    boPin141ToolValue := boPin141.Value;

                  
END_GET
END_PROPERTY

PROPERTY boPin122ToolValue : BOOL
GET
                    boPin122ToolValue := boPin122.Value;

                  
END_GET
END_PROPERTY

PROPERTY boPin146ToolValue : BOOL
GET
                    boPin146ToolValue := boPin146.Value;

                  
END_GET
END_PROPERTY

PROPERTY boPin123ToolValue : BOOL
GET
                    boPin123ToolValue := boPin123.Value;

                  
END_GET
END_PROPERTY

PROPERTY boPin187ToolValue : BOOL
GET
                    boPin187ToolValue := boPin187.Value;

                  
END_GET
END_PROPERTY

PROPERTY boPin124ToolValue : BOOL
GET
                    boPin124ToolValue := boPin124.Value;

                  
END_GET
END_PROPERTY

PROPERTY boPin148ToolValue : BOOL
GET
                    boPin148ToolValue := boPin148.Value;

                  
END_GET
END_PROPERTY

PROPERTY boPin153ToolValue : BOOL
GET
                    boPin153ToolValue := boPin153.Value;

                  
END_GET
END_PROPERTY

PROPERTY boPin177ToolValue : BOOL
GET
                    boPin177ToolValue := boPin177.Value;

                  
END_GET
END_PROPERTY

PROPERTY boPin156ToolValue : BOOL
GET
                    boPin156ToolValue := boPin156.Value;

                  
END_GET
END_PROPERTY

PROPERTY boPin159ToolValue : BOOL
GET
                    boPin159ToolValue := boPin159.Value;

                  
END_GET
END_PROPERTY

PROPERTY boPin186ToolValue : BOOL
GET
                    boPin186ToolValue := boPin186.Value;

                  
END_GET
END_PROPERTY

PROPERTY boPin162ToolValue : BOOL
GET
                    boPin162ToolValue := boPin162.Value;

                  
END_GET
END_PROPERTY

PROPERTY boPin189ToolValue : BOOL
GET
                    boPin189ToolValue := boPin189.Value;

                  
END_GET
END_PROPERTY

PROPERTY boPin165ToolValue : BOOL
GET
                    boPin165ToolValue := boPin165.Value;

                  
END_GET
END_PROPERTY

PROPERTY boPin195ToolValue : BOOL
GET
                    boPin195ToolValue := boPin195.Value;

                  
END_GET
END_PROPERTY

PROPERTY boPin171ToolValue : BOOL
GET
                    boPin171ToolValue := boPin171.Value;

                  
END_GET
END_PROPERTY

PROPERTY boPin154ToolValue : BOOL
GET
                    boPin154ToolValue := boPin154.Value;

                  
END_GET
END_PROPERTY

PROPERTY boPin160ToolValue : BOOL
GET
                    boPin160ToolValue := boPin160.Value;

                  
END_GET
END_PROPERTY

PROPERTY boPin184ToolValue : BOOL
GET
                    boPin184ToolValue := boPin184.Value;

                  
END_GET
END_PROPERTY

PROPERTY boPin163ToolValue : BOOL
GET
                    boPin163ToolValue := boPin163.Value;

                  
END_GET
END_PROPERTY

PROPERTY boPin190ToolValue : BOOL
GET
                    boPin190ToolValue := boPin190.Value;

                  
END_GET
END_PROPERTY

PROPERTY boPin166ToolValue : BOOL
GET
                    boPin166ToolValue := boPin166.Value;

                  
END_GET
END_PROPERTY

PROPERTY boPin193ToolValue : BOOL
GET
                    boPin193ToolValue := boPin193.Value;

                  
END_GET
END_PROPERTY

PROPERTY boPin169ToolValue : BOOL
GET
                    boPin169ToolValue := boPin169.Value;

                  
END_GET
END_PROPERTY

PROPERTY boPin196ToolValue : BOOL
GET
                    boPin196ToolValue := boPin196.Value;

                  
END_GET
END_PROPERTY

PROPERTY boPin172ToolValue : BOOL
GET
                    boPin172ToolValue := boPin172.Value;

                  
END_GET
END_PROPERTY

PROPERTY boPin149ToolValue : BOOL
GET
                    boPin149ToolValue := boPin149.Value;

                  
END_GET
END_PROPERTY

PROPERTY boPin173ToolValue : BOOL
GET
                    boPin173ToolValue := boPin173.Value;

                  
END_GET
END_PROPERTY

PROPERTY boPin152ToolValue : BOOL
GET
                    boPin152ToolValue := boPin152.Value;

                  
END_GET
END_PROPERTY

PROPERTY boPin176ToolValue : BOOL
GET
                    boPin176ToolValue := boPin176.Value;

                  
END_GET
END_PROPERTY

PROPERTY boPin155ToolValue : BOOL
GET
                    boPin155ToolValue := boPin155.Value;

                  
END_GET
END_PROPERTY

PROPERTY boPin179ToolValue : BOOL
GET
                    boPin179ToolValue := boPin179.Value;

                  
END_GET
END_PROPERTY

PROPERTY boPin158ToolValue : BOOL
GET
                    boPin158ToolValue := boPin158.Value;

                  
END_GET
END_PROPERTY

PROPERTY boPin182ToolValue : BOOL
GET
                    boPin182ToolValue := boPin182.Value;

                  
END_GET
END_PROPERTY

PROPERTY boPin252ToolValue : BOOL
GET
                    boPin252ToolValue := boPin252.Value;

                  
END_GET
END_PROPERTY

PROPERTY boPin239ToolValue : BOOL
GET
                    boPin239ToolValue := boPin239.Value;

                  
END_GET
END_PROPERTY

PROPERTY boPin188ToolValue : BOOL
GET
                    boPin188ToolValue := boPin188.Value;

                  
END_GET
END_PROPERTY

PROPERTY boPin164ToolValue : BOOL
GET
                    boPin164ToolValue := boPin164.Value;

                  
END_GET
END_PROPERTY

PROPERTY boPin191ToolValue : BOOL
GET
                    boPin191ToolValue := boPin191.Value;

                  
END_GET
END_PROPERTY

PROPERTY boPin167ToolValue : BOOL
GET
                    boPin167ToolValue := boPin167.Value;

                  
END_GET
END_PROPERTY

PROPERTY boPin194ToolValue : BOOL
GET
                    boPin194ToolValue := boPin194.Value;

                  
END_GET
END_PROPERTY

PROPERTY boPin170ToolValue : BOOL
GET
                    boPin170ToolValue := boPin170.Value;

                  
END_GET
END_PROPERTY

PROPERTY boPin192ToolValue : BOOL
GET
                    boPin192ToolValue := boPin192.Value;

                  
END_GET
END_PROPERTY

PROPERTY boPin168ToolValue : BOOL
GET
                    boPin168ToolValue := boPin168.Value;

                  
END_GET
END_PROPERTY

METHOD InitializeCanSignals
                  boPin107.AppScalingDivisor :=1;
boPin107.AppScalingMultiplier :=1;
boPin107.AppScalingOffset :=0;
boPin107.AppUnit :="";
boPin107.CanDefault :=0;
boPin107.CanInit :=0;
boPin107.CanMax :=1;
boPin107.CanMin :=0;
boPin107.CanUnit :="";
boPin107.Description :="for the Neotec diag pages";
boPin107.ErrorReaction := eErrorReaction.ERSIG_DFLT;
boPin107.ReceiverAdress :=1;
boPin107.ToolScalingDivisor :=1;
boPin107.ToolScalingMultiplier :=1;
boPin107.ToolScalingOffset :=0;
boPin107.ToolUnit :="";

boPin131.AppScalingDivisor :=1;
boPin131.AppScalingMultiplier :=1;
boPin131.AppScalingOffset :=0;
boPin131.AppUnit :="";
boPin131.CanDefault :=0;
boPin131.CanInit :=0;
boPin131.CanMax :=1;
boPin131.CanMin :=0;
boPin131.CanUnit :="";
boPin131.Description :="for the Neotec diag pages";
boPin131.ErrorReaction := eErrorReaction.ERSIG_DFLT;
boPin131.ReceiverAdress :=1;
boPin131.ToolScalingDivisor :=1;
boPin131.ToolScalingMultiplier :=1;
boPin131.ToolScalingOffset :=0;
boPin131.ToolUnit :="";

boPin108.AppScalingDivisor :=1;
boPin108.AppScalingMultiplier :=1;
boPin108.AppScalingOffset :=0;
boPin108.AppUnit :="";
boPin108.CanDefault :=0;
boPin108.CanInit :=0;
boPin108.CanMax :=1;
boPin108.CanMin :=0;
boPin108.CanUnit :="";
boPin108.Description :="for the Neotec diag pages";
boPin108.ErrorReaction := eErrorReaction.ERSIG_DFLT;
boPin108.ReceiverAdress :=1;
boPin108.ToolScalingDivisor :=1;
boPin108.ToolScalingMultiplier :=1;
boPin108.ToolScalingOffset :=0;
boPin108.ToolUnit :="";

boPin132.AppScalingDivisor :=1;
boPin132.AppScalingMultiplier :=1;
boPin132.AppScalingOffset :=0;
boPin132.AppUnit :="";
boPin132.CanDefault :=0;
boPin132.CanInit :=0;
boPin132.CanMax :=1;
boPin132.CanMin :=0;
boPin132.CanUnit :="";
boPin132.Description :="for the Neotec diag pages";
boPin132.ErrorReaction := eErrorReaction.ERSIG_DFLT;
boPin132.ReceiverAdress :=1;
boPin132.ToolScalingDivisor :=1;
boPin132.ToolScalingMultiplier :=1;
boPin132.ToolScalingOffset :=0;
boPin132.ToolUnit :="";

boPin109.AppScalingDivisor :=1;
boPin109.AppScalingMultiplier :=1;
boPin109.AppScalingOffset :=0;
boPin109.AppUnit :="";
boPin109.CanDefault :=0;
boPin109.CanInit :=0;
boPin109.CanMax :=1;
boPin109.CanMin :=0;
boPin109.CanUnit :="";
boPin109.Description :="for the Neotec diag pages";
boPin109.ErrorReaction := eErrorReaction.ERSIG_DFLT;
boPin109.ReceiverAdress :=1;
boPin109.ToolScalingDivisor :=1;
boPin109.ToolScalingMultiplier :=1;
boPin109.ToolScalingOffset :=0;
boPin109.ToolUnit :="";

boPin133.AppScalingDivisor :=1;
boPin133.AppScalingMultiplier :=1;
boPin133.AppScalingOffset :=0;
boPin133.AppUnit :="";
boPin133.CanDefault :=0;
boPin133.CanInit :=0;
boPin133.CanMax :=1;
boPin133.CanMin :=0;
boPin133.CanUnit :="";
boPin133.Description :="for the Neotec diag pages";
boPin133.ErrorReaction := eErrorReaction.ERSIG_DFLT;
boPin133.ReceiverAdress :=1;
boPin133.ToolScalingDivisor :=1;
boPin133.ToolScalingMultiplier :=1;
boPin133.ToolScalingOffset :=0;
boPin133.ToolUnit :="";

boPin110.AppScalingDivisor :=1;
boPin110.AppScalingMultiplier :=1;
boPin110.AppScalingOffset :=0;
boPin110.AppUnit :="";
boPin110.CanDefault :=0;
boPin110.CanInit :=0;
boPin110.CanMax :=1;
boPin110.CanMin :=0;
boPin110.CanUnit :="";
boPin110.Description :="for the Neotec diag pages";
boPin110.ErrorReaction := eErrorReaction.ERSIG_DFLT;
boPin110.ReceiverAdress :=1;
boPin110.ToolScalingDivisor :=1;
boPin110.ToolScalingMultiplier :=1;
boPin110.ToolScalingOffset :=0;
boPin110.ToolUnit :="";

boPin134.AppScalingDivisor :=1;
boPin134.AppScalingMultiplier :=1;
boPin134.AppScalingOffset :=0;
boPin134.AppUnit :="";
boPin134.CanDefault :=0;
boPin134.CanInit :=0;
boPin134.CanMax :=1;
boPin134.CanMin :=0;
boPin134.CanUnit :="";
boPin134.Description :="for the Neotec diag pages";
boPin134.ErrorReaction := eErrorReaction.ERSIG_DFLT;
boPin134.ReceiverAdress :=1;
boPin134.ToolScalingDivisor :=1;
boPin134.ToolScalingMultiplier :=1;
boPin134.ToolScalingOffset :=0;
boPin134.ToolUnit :="";

boPin111.AppScalingDivisor :=1;
boPin111.AppScalingMultiplier :=1;
boPin111.AppScalingOffset :=0;
boPin111.AppUnit :="";
boPin111.CanDefault :=0;
boPin111.CanInit :=0;
boPin111.CanMax :=1;
boPin111.CanMin :=0;
boPin111.CanUnit :="";
boPin111.Description :="for the Neotec diag pages";
boPin111.ErrorReaction := eErrorReaction.ERSIG_DFLT;
boPin111.ReceiverAdress :=1;
boPin111.ToolScalingDivisor :=1;
boPin111.ToolScalingMultiplier :=1;
boPin111.ToolScalingOffset :=0;
boPin111.ToolUnit :="";

boPin135.AppScalingDivisor :=1;
boPin135.AppScalingMultiplier :=1;
boPin135.AppScalingOffset :=0;
boPin135.AppUnit :="";
boPin135.CanDefault :=0;
boPin135.CanInit :=0;
boPin135.CanMax :=1;
boPin135.CanMin :=0;
boPin135.CanUnit :="";
boPin135.Description :="for the Neotec diag pages";
boPin135.ErrorReaction := eErrorReaction.ERSIG_DFLT;
boPin135.ReceiverAdress :=1;
boPin135.ToolScalingDivisor :=1;
boPin135.ToolScalingMultiplier :=1;
boPin135.ToolScalingOffset :=0;
boPin135.ToolUnit :="";

boPin112.AppScalingDivisor :=1;
boPin112.AppScalingMultiplier :=1;
boPin112.AppScalingOffset :=0;
boPin112.AppUnit :="";
boPin112.CanDefault :=0;
boPin112.CanInit :=0;
boPin112.CanMax :=1;
boPin112.CanMin :=0;
boPin112.CanUnit :="";
boPin112.Description :="for the Neotec diag pages";
boPin112.ErrorReaction := eErrorReaction.ERSIG_DFLT;
boPin112.ReceiverAdress :=1;
boPin112.ToolScalingDivisor :=1;
boPin112.ToolScalingMultiplier :=1;
boPin112.ToolScalingOffset :=0;
boPin112.ToolUnit :="";

boPin136.AppScalingDivisor :=1;
boPin136.AppScalingMultiplier :=1;
boPin136.AppScalingOffset :=0;
boPin136.AppUnit :="";
boPin136.CanDefault :=0;
boPin136.CanInit :=0;
boPin136.CanMax :=1;
boPin136.CanMin :=0;
boPin136.CanUnit :="";
boPin136.Description :="for the Neotec diag pages";
boPin136.ErrorReaction := eErrorReaction.ERSIG_DFLT;
boPin136.ReceiverAdress :=1;
boPin136.ToolScalingDivisor :=1;
boPin136.ToolScalingMultiplier :=1;
boPin136.ToolScalingOffset :=0;
boPin136.ToolUnit :="";

boPin113.AppScalingDivisor :=1;
boPin113.AppScalingMultiplier :=1;
boPin113.AppScalingOffset :=0;
boPin113.AppUnit :="";
boPin113.CanDefault :=0;
boPin113.CanInit :=0;
boPin113.CanMax :=1;
boPin113.CanMin :=0;
boPin113.CanUnit :="";
boPin113.Description :="for the Neotec diag pages";
boPin113.ErrorReaction := eErrorReaction.ERSIG_DFLT;
boPin113.ReceiverAdress :=1;
boPin113.ToolScalingDivisor :=1;
boPin113.ToolScalingMultiplier :=1;
boPin113.ToolScalingOffset :=0;
boPin113.ToolUnit :="";

boPin137.AppScalingDivisor :=1;
boPin137.AppScalingMultiplier :=1;
boPin137.AppScalingOffset :=0;
boPin137.AppUnit :="";
boPin137.CanDefault :=0;
boPin137.CanInit :=0;
boPin137.CanMax :=1;
boPin137.CanMin :=0;
boPin137.CanUnit :="";
boPin137.Description :="for the Neotec diag pages";
boPin137.ErrorReaction := eErrorReaction.ERSIG_DFLT;
boPin137.ReceiverAdress :=1;
boPin137.ToolScalingDivisor :=1;
boPin137.ToolScalingMultiplier :=1;
boPin137.ToolScalingOffset :=0;
boPin137.ToolUnit :="";

boPin114.AppScalingDivisor :=1;
boPin114.AppScalingMultiplier :=1;
boPin114.AppScalingOffset :=0;
boPin114.AppUnit :="";
boPin114.CanDefault :=0;
boPin114.CanInit :=0;
boPin114.CanMax :=1;
boPin114.CanMin :=0;
boPin114.CanUnit :="";
boPin114.Description :="for the Neotec diag pages";
boPin114.ErrorReaction := eErrorReaction.ERSIG_DFLT;
boPin114.ReceiverAdress :=1;
boPin114.ToolScalingDivisor :=1;
boPin114.ToolScalingMultiplier :=1;
boPin114.ToolScalingOffset :=0;
boPin114.ToolUnit :="";

boPin138.AppScalingDivisor :=1;
boPin138.AppScalingMultiplier :=1;
boPin138.AppScalingOffset :=0;
boPin138.AppUnit :="";
boPin138.CanDefault :=0;
boPin138.CanInit :=0;
boPin138.CanMax :=1;
boPin138.CanMin :=0;
boPin138.CanUnit :="";
boPin138.Description :="for the Neotec diag pages";
boPin138.ErrorReaction := eErrorReaction.ERSIG_DFLT;
boPin138.ReceiverAdress :=1;
boPin138.ToolScalingDivisor :=1;
boPin138.ToolScalingMultiplier :=1;
boPin138.ToolScalingOffset :=0;
boPin138.ToolUnit :="";

boPin140.AppScalingDivisor :=1;
boPin140.AppScalingMultiplier :=1;
boPin140.AppScalingOffset :=0;
boPin140.AppUnit :="";
boPin140.CanDefault :=0;
boPin140.CanInit :=0;
boPin140.CanMax :=1;
boPin140.CanMin :=0;
boPin140.CanUnit :="";
boPin140.Description :="for the Neotec diag pages";
boPin140.ErrorReaction := eErrorReaction.ERSIG_DFLT;
boPin140.ReceiverAdress :=1;
boPin140.ToolScalingDivisor :=1;
boPin140.ToolScalingMultiplier :=1;
boPin140.ToolScalingOffset :=0;
boPin140.ToolUnit :="";

boPin117.AppScalingDivisor :=1;
boPin117.AppScalingMultiplier :=1;
boPin117.AppScalingOffset :=0;
boPin117.AppUnit :="";
boPin117.CanDefault :=0;
boPin117.CanInit :=0;
boPin117.CanMax :=1;
boPin117.CanMin :=0;
boPin117.CanUnit :="";
boPin117.Description :="for the Neotec diag pages";
boPin117.ErrorReaction := eErrorReaction.ERSIG_DFLT;
boPin117.ReceiverAdress :=1;
boPin117.ToolScalingDivisor :=1;
boPin117.ToolScalingMultiplier :=1;
boPin117.ToolScalingOffset :=0;
boPin117.ToolUnit :="";

boPin141.AppScalingDivisor :=1;
boPin141.AppScalingMultiplier :=1;
boPin141.AppScalingOffset :=0;
boPin141.AppUnit :="";
boPin141.CanDefault :=0;
boPin141.CanInit :=0;
boPin141.CanMax :=1;
boPin141.CanMin :=0;
boPin141.CanUnit :="";
boPin141.Description :="for the Neotec diag pages";
boPin141.ErrorReaction := eErrorReaction.ERSIG_DFLT;
boPin141.ReceiverAdress :=1;
boPin141.ToolScalingDivisor :=1;
boPin141.ToolScalingMultiplier :=1;
boPin141.ToolScalingOffset :=0;
boPin141.ToolUnit :="";

boPin122.AppScalingDivisor :=1;
boPin122.AppScalingMultiplier :=1;
boPin122.AppScalingOffset :=0;
boPin122.AppUnit :="";
boPin122.CanDefault :=0;
boPin122.CanInit :=0;
boPin122.CanMax :=1;
boPin122.CanMin :=0;
boPin122.CanUnit :="";
boPin122.Description :="for the Neotec diag pages";
boPin122.ErrorReaction := eErrorReaction.ERSIG_DFLT;
boPin122.ReceiverAdress :=1;
boPin122.ToolScalingDivisor :=1;
boPin122.ToolScalingMultiplier :=1;
boPin122.ToolScalingOffset :=0;
boPin122.ToolUnit :="";

boPin146.AppScalingDivisor :=1;
boPin146.AppScalingMultiplier :=1;
boPin146.AppScalingOffset :=0;
boPin146.AppUnit :="";
boPin146.CanDefault :=0;
boPin146.CanInit :=0;
boPin146.CanMax :=1;
boPin146.CanMin :=0;
boPin146.CanUnit :="";
boPin146.Description :="for the Neotec diag pages";
boPin146.ErrorReaction := eErrorReaction.ERSIG_DFLT;
boPin146.ReceiverAdress :=1;
boPin146.ToolScalingDivisor :=1;
boPin146.ToolScalingMultiplier :=1;
boPin146.ToolScalingOffset :=0;
boPin146.ToolUnit :="";

boPin123.AppScalingDivisor :=1;
boPin123.AppScalingMultiplier :=1;
boPin123.AppScalingOffset :=0;
boPin123.AppUnit :="";
boPin123.CanDefault :=0;
boPin123.CanInit :=0;
boPin123.CanMax :=1;
boPin123.CanMin :=0;
boPin123.CanUnit :="";
boPin123.Description :="for the Neotec diag pages";
boPin123.ErrorReaction := eErrorReaction.ERSIG_DFLT;
boPin123.ReceiverAdress :=1;
boPin123.ToolScalingDivisor :=1;
boPin123.ToolScalingMultiplier :=1;
boPin123.ToolScalingOffset :=0;
boPin123.ToolUnit :="";

boPin187.AppScalingDivisor :=1;
boPin187.AppScalingMultiplier :=1;
boPin187.AppScalingOffset :=0;
boPin187.AppUnit :="";
boPin187.CanDefault :=0;
boPin187.CanInit :=0;
boPin187.CanMax :=1;
boPin187.CanMin :=0;
boPin187.CanUnit :="";
boPin187.Description :="for the Neotec diag pages";
boPin187.ErrorReaction := eErrorReaction.ERSIG_DFLT;
boPin187.ReceiverAdress :=1;
boPin187.ToolScalingDivisor :=1;
boPin187.ToolScalingMultiplier :=1;
boPin187.ToolScalingOffset :=0;
boPin187.ToolUnit :="";

boPin124.AppScalingDivisor :=1;
boPin124.AppScalingMultiplier :=1;
boPin124.AppScalingOffset :=0;
boPin124.AppUnit :="";
boPin124.CanDefault :=0;
boPin124.CanInit :=0;
boPin124.CanMax :=1;
boPin124.CanMin :=0;
boPin124.CanUnit :="";
boPin124.Description :="for the Neotec diag pages";
boPin124.ErrorReaction := eErrorReaction.ERSIG_DFLT;
boPin124.ReceiverAdress :=1;
boPin124.ToolScalingDivisor :=1;
boPin124.ToolScalingMultiplier :=1;
boPin124.ToolScalingOffset :=0;
boPin124.ToolUnit :="";

boPin148.AppScalingDivisor :=1;
boPin148.AppScalingMultiplier :=1;
boPin148.AppScalingOffset :=0;
boPin148.AppUnit :="";
boPin148.CanDefault :=0;
boPin148.CanInit :=0;
boPin148.CanMax :=1;
boPin148.CanMin :=0;
boPin148.CanUnit :="";
boPin148.Description :="for the Neotec diag pages";
boPin148.ErrorReaction := eErrorReaction.ERSIG_DFLT;
boPin148.ReceiverAdress :=1;
boPin148.ToolScalingDivisor :=1;
boPin148.ToolScalingMultiplier :=1;
boPin148.ToolScalingOffset :=0;
boPin148.ToolUnit :="";

boPin153.AppScalingDivisor :=1;
boPin153.AppScalingMultiplier :=1;
boPin153.AppScalingOffset :=0;
boPin153.AppUnit :="";
boPin153.CanDefault :=0;
boPin153.CanInit :=0;
boPin153.CanMax :=1;
boPin153.CanMin :=0;
boPin153.CanUnit :="";
boPin153.Description :="for the Neotec diag pages";
boPin153.ErrorReaction := eErrorReaction.ERSIG_DFLT;
boPin153.ReceiverAdress :=1;
boPin153.ToolScalingDivisor :=1;
boPin153.ToolScalingMultiplier :=1;
boPin153.ToolScalingOffset :=0;
boPin153.ToolUnit :="";

boPin177.AppScalingDivisor :=1;
boPin177.AppScalingMultiplier :=1;
boPin177.AppScalingOffset :=0;
boPin177.AppUnit :="";
boPin177.CanDefault :=0;
boPin177.CanInit :=0;
boPin177.CanMax :=1;
boPin177.CanMin :=0;
boPin177.CanUnit :="";
boPin177.Description :="for the Neotec diag pages";
boPin177.ErrorReaction := eErrorReaction.ERSIG_DFLT;
boPin177.ReceiverAdress :=1;
boPin177.ToolScalingDivisor :=1;
boPin177.ToolScalingMultiplier :=1;
boPin177.ToolScalingOffset :=0;
boPin177.ToolUnit :="";

boPin156.AppScalingDivisor :=1;
boPin156.AppScalingMultiplier :=1;
boPin156.AppScalingOffset :=0;
boPin156.AppUnit :="";
boPin156.CanDefault :=0;
boPin156.CanInit :=0;
boPin156.CanMax :=1;
boPin156.CanMin :=0;
boPin156.CanUnit :="";
boPin156.Description :="for the Neotec diag pages";
boPin156.ErrorReaction := eErrorReaction.ERSIG_DFLT;
boPin156.ReceiverAdress :=1;
boPin156.ToolScalingDivisor :=1;
boPin156.ToolScalingMultiplier :=1;
boPin156.ToolScalingOffset :=0;
boPin156.ToolUnit :="";

boPin159.AppScalingDivisor :=1;
boPin159.AppScalingMultiplier :=1;
boPin159.AppScalingOffset :=0;
boPin159.AppUnit :="";
boPin159.CanDefault :=0;
boPin159.CanInit :=0;
boPin159.CanMax :=1;
boPin159.CanMin :=0;
boPin159.CanUnit :="";
boPin159.Description :="for the Neotec diag pages";
boPin159.ErrorReaction := eErrorReaction.ERSIG_DFLT;
boPin159.ReceiverAdress :=1;
boPin159.ToolScalingDivisor :=1;
boPin159.ToolScalingMultiplier :=1;
boPin159.ToolScalingOffset :=0;
boPin159.ToolUnit :="";

boPin186.AppScalingDivisor :=1;
boPin186.AppScalingMultiplier :=1;
boPin186.AppScalingOffset :=0;
boPin186.AppUnit :="";
boPin186.CanDefault :=0;
boPin186.CanInit :=0;
boPin186.CanMax :=1;
boPin186.CanMin :=0;
boPin186.CanUnit :="";
boPin186.Description :="for the Neotec diag pages";
boPin186.ErrorReaction := eErrorReaction.ERSIG_DFLT;
boPin186.ReceiverAdress :=1;
boPin186.ToolScalingDivisor :=1;
boPin186.ToolScalingMultiplier :=1;
boPin186.ToolScalingOffset :=0;
boPin186.ToolUnit :="";

boPin162.AppScalingDivisor :=1;
boPin162.AppScalingMultiplier :=1;
boPin162.AppScalingOffset :=0;
boPin162.AppUnit :="";
boPin162.CanDefault :=0;
boPin162.CanInit :=0;
boPin162.CanMax :=1;
boPin162.CanMin :=0;
boPin162.CanUnit :="";
boPin162.Description :="for the Neotec diag pages";
boPin162.ErrorReaction := eErrorReaction.ERSIG_DFLT;
boPin162.ReceiverAdress :=1;
boPin162.ToolScalingDivisor :=1;
boPin162.ToolScalingMultiplier :=1;
boPin162.ToolScalingOffset :=0;
boPin162.ToolUnit :="";

boPin189.AppScalingDivisor :=1;
boPin189.AppScalingMultiplier :=1;
boPin189.AppScalingOffset :=0;
boPin189.AppUnit :="";
boPin189.CanDefault :=0;
boPin189.CanInit :=0;
boPin189.CanMax :=1;
boPin189.CanMin :=0;
boPin189.CanUnit :="";
boPin189.Description :="for the Neotec diag pages";
boPin189.ErrorReaction := eErrorReaction.ERSIG_DFLT;
boPin189.ReceiverAdress :=1;
boPin189.ToolScalingDivisor :=1;
boPin189.ToolScalingMultiplier :=1;
boPin189.ToolScalingOffset :=0;
boPin189.ToolUnit :="";

boPin165.AppScalingDivisor :=1;
boPin165.AppScalingMultiplier :=1;
boPin165.AppScalingOffset :=0;
boPin165.AppUnit :="";
boPin165.CanDefault :=0;
boPin165.CanInit :=0;
boPin165.CanMax :=1;
boPin165.CanMin :=0;
boPin165.CanUnit :="";
boPin165.Description :="for the Neotec diag pages";
boPin165.ErrorReaction := eErrorReaction.ERSIG_DFLT;
boPin165.ReceiverAdress :=1;
boPin165.ToolScalingDivisor :=1;
boPin165.ToolScalingMultiplier :=1;
boPin165.ToolScalingOffset :=0;
boPin165.ToolUnit :="";

boPin195.AppScalingDivisor :=1;
boPin195.AppScalingMultiplier :=1;
boPin195.AppScalingOffset :=0;
boPin195.AppUnit :="";
boPin195.CanDefault :=0;
boPin195.CanInit :=0;
boPin195.CanMax :=1;
boPin195.CanMin :=0;
boPin195.CanUnit :="";
boPin195.Description :="for the Neotec diag pages";
boPin195.ErrorReaction := eErrorReaction.ERSIG_DFLT;
boPin195.ReceiverAdress :=1;
boPin195.ToolScalingDivisor :=1;
boPin195.ToolScalingMultiplier :=1;
boPin195.ToolScalingOffset :=0;
boPin195.ToolUnit :="";

boPin171.AppScalingDivisor :=1;
boPin171.AppScalingMultiplier :=1;
boPin171.AppScalingOffset :=0;
boPin171.AppUnit :="";
boPin171.CanDefault :=0;
boPin171.CanInit :=0;
boPin171.CanMax :=1;
boPin171.CanMin :=0;
boPin171.CanUnit :="";
boPin171.Description :="for the Neotec diag pages";
boPin171.ErrorReaction := eErrorReaction.ERSIG_DFLT;
boPin171.ReceiverAdress :=1;
boPin171.ToolScalingDivisor :=1;
boPin171.ToolScalingMultiplier :=1;
boPin171.ToolScalingOffset :=0;
boPin171.ToolUnit :="";

boPin154.AppScalingDivisor :=1;
boPin154.AppScalingMultiplier :=1;
boPin154.AppScalingOffset :=0;
boPin154.AppUnit :="";
boPin154.CanDefault :=0;
boPin154.CanInit :=0;
boPin154.CanMax :=1;
boPin154.CanMin :=0;
boPin154.CanUnit :="";
boPin154.Description :="for the Neotec diag pages";
boPin154.ErrorReaction := eErrorReaction.ERSIG_DFLT;
boPin154.ReceiverAdress :=1;
boPin154.ToolScalingDivisor :=1;
boPin154.ToolScalingMultiplier :=1;
boPin154.ToolScalingOffset :=0;
boPin154.ToolUnit :="";

boPin160.AppScalingDivisor :=1;
boPin160.AppScalingMultiplier :=1;
boPin160.AppScalingOffset :=0;
boPin160.AppUnit :="";
boPin160.CanDefault :=0;
boPin160.CanInit :=0;
boPin160.CanMax :=1;
boPin160.CanMin :=0;
boPin160.CanUnit :="";
boPin160.Description :="for the Neotec diag pages";
boPin160.ErrorReaction := eErrorReaction.ERSIG_DFLT;
boPin160.ReceiverAdress :=1;
boPin160.ToolScalingDivisor :=1;
boPin160.ToolScalingMultiplier :=1;
boPin160.ToolScalingOffset :=0;
boPin160.ToolUnit :="";

boPin184.AppScalingDivisor :=1;
boPin184.AppScalingMultiplier :=1;
boPin184.AppScalingOffset :=0;
boPin184.AppUnit :="";
boPin184.CanDefault :=0;
boPin184.CanInit :=0;
boPin184.CanMax :=1;
boPin184.CanMin :=0;
boPin184.CanUnit :="";
boPin184.Description :="for the Neotec diag pages";
boPin184.ErrorReaction := eErrorReaction.ERSIG_DFLT;
boPin184.ReceiverAdress :=1;
boPin184.ToolScalingDivisor :=1;
boPin184.ToolScalingMultiplier :=1;
boPin184.ToolScalingOffset :=0;
boPin184.ToolUnit :="";

boPin163.AppScalingDivisor :=1;
boPin163.AppScalingMultiplier :=1;
boPin163.AppScalingOffset :=0;
boPin163.AppUnit :="";
boPin163.CanDefault :=0;
boPin163.CanInit :=0;
boPin163.CanMax :=1;
boPin163.CanMin :=0;
boPin163.CanUnit :="";
boPin163.Description :="for the Neotec diag pages";
boPin163.ErrorReaction := eErrorReaction.ERSIG_DFLT;
boPin163.ReceiverAdress :=1;
boPin163.ToolScalingDivisor :=1;
boPin163.ToolScalingMultiplier :=1;
boPin163.ToolScalingOffset :=0;
boPin163.ToolUnit :="";

boPin190.AppScalingDivisor :=1;
boPin190.AppScalingMultiplier :=1;
boPin190.AppScalingOffset :=0;
boPin190.AppUnit :="";
boPin190.CanDefault :=0;
boPin190.CanInit :=0;
boPin190.CanMax :=1;
boPin190.CanMin :=0;
boPin190.CanUnit :="";
boPin190.Description :="for the Neotec diag pages";
boPin190.ErrorReaction := eErrorReaction.ERSIG_DFLT;
boPin190.ReceiverAdress :=1;
boPin190.ToolScalingDivisor :=1;
boPin190.ToolScalingMultiplier :=1;
boPin190.ToolScalingOffset :=0;
boPin190.ToolUnit :="";

boPin166.AppScalingDivisor :=1;
boPin166.AppScalingMultiplier :=1;
boPin166.AppScalingOffset :=0;
boPin166.AppUnit :="";
boPin166.CanDefault :=0;
boPin166.CanInit :=0;
boPin166.CanMax :=1;
boPin166.CanMin :=0;
boPin166.CanUnit :="";
boPin166.Description :="for the Neotec diag pages";
boPin166.ErrorReaction := eErrorReaction.ERSIG_DFLT;
boPin166.ReceiverAdress :=1;
boPin166.ToolScalingDivisor :=1;
boPin166.ToolScalingMultiplier :=1;
boPin166.ToolScalingOffset :=0;
boPin166.ToolUnit :="";

boPin193.AppScalingDivisor :=1;
boPin193.AppScalingMultiplier :=1;
boPin193.AppScalingOffset :=0;
boPin193.AppUnit :="";
boPin193.CanDefault :=0;
boPin193.CanInit :=0;
boPin193.CanMax :=1;
boPin193.CanMin :=0;
boPin193.CanUnit :="";
boPin193.Description :="for the Neotec diag pages";
boPin193.ErrorReaction := eErrorReaction.ERSIG_DFLT;
boPin193.ReceiverAdress :=1;
boPin193.ToolScalingDivisor :=1;
boPin193.ToolScalingMultiplier :=1;
boPin193.ToolScalingOffset :=0;
boPin193.ToolUnit :="";

boPin169.AppScalingDivisor :=1;
boPin169.AppScalingMultiplier :=1;
boPin169.AppScalingOffset :=0;
boPin169.AppUnit :="";
boPin169.CanDefault :=0;
boPin169.CanInit :=0;
boPin169.CanMax :=1;
boPin169.CanMin :=0;
boPin169.CanUnit :="";
boPin169.Description :="for the Neotec diag pages";
boPin169.ErrorReaction := eErrorReaction.ERSIG_DFLT;
boPin169.ReceiverAdress :=1;
boPin169.ToolScalingDivisor :=1;
boPin169.ToolScalingMultiplier :=1;
boPin169.ToolScalingOffset :=0;
boPin169.ToolUnit :="";

boPin196.AppScalingDivisor :=1;
boPin196.AppScalingMultiplier :=1;
boPin196.AppScalingOffset :=0;
boPin196.AppUnit :="";
boPin196.CanDefault :=0;
boPin196.CanInit :=0;
boPin196.CanMax :=1;
boPin196.CanMin :=0;
boPin196.CanUnit :="";
boPin196.Description :="for the Neotec diag pages";
boPin196.ErrorReaction := eErrorReaction.ERSIG_DFLT;
boPin196.ReceiverAdress :=1;
boPin196.ToolScalingDivisor :=1;
boPin196.ToolScalingMultiplier :=1;
boPin196.ToolScalingOffset :=0;
boPin196.ToolUnit :="";

boPin172.AppScalingDivisor :=1;
boPin172.AppScalingMultiplier :=1;
boPin172.AppScalingOffset :=0;
boPin172.AppUnit :="";
boPin172.CanDefault :=0;
boPin172.CanInit :=0;
boPin172.CanMax :=1;
boPin172.CanMin :=0;
boPin172.CanUnit :="";
boPin172.Description :="for the Neotec diag pages";
boPin172.ErrorReaction := eErrorReaction.ERSIG_DFLT;
boPin172.ReceiverAdress :=1;
boPin172.ToolScalingDivisor :=1;
boPin172.ToolScalingMultiplier :=1;
boPin172.ToolScalingOffset :=0;
boPin172.ToolUnit :="";

boPin149.AppScalingDivisor :=1;
boPin149.AppScalingMultiplier :=1;
boPin149.AppScalingOffset :=0;
boPin149.AppUnit :="";
boPin149.CanDefault :=0;
boPin149.CanInit :=0;
boPin149.CanMax :=1;
boPin149.CanMin :=0;
boPin149.CanUnit :="";
boPin149.Description :="for the Neotec diag pages";
boPin149.ErrorReaction := eErrorReaction.ERSIG_DFLT;
boPin149.ReceiverAdress :=1;
boPin149.ToolScalingDivisor :=1;
boPin149.ToolScalingMultiplier :=1;
boPin149.ToolScalingOffset :=0;
boPin149.ToolUnit :="";

boPin173.AppScalingDivisor :=1;
boPin173.AppScalingMultiplier :=1;
boPin173.AppScalingOffset :=0;
boPin173.AppUnit :="";
boPin173.CanDefault :=0;
boPin173.CanInit :=0;
boPin173.CanMax :=1;
boPin173.CanMin :=0;
boPin173.CanUnit :="";
boPin173.Description :="for the Neotec diag pages";
boPin173.ErrorReaction := eErrorReaction.ERSIG_DFLT;
boPin173.ReceiverAdress :=1;
boPin173.ToolScalingDivisor :=1;
boPin173.ToolScalingMultiplier :=1;
boPin173.ToolScalingOffset :=0;
boPin173.ToolUnit :="";

boPin152.AppScalingDivisor :=1;
boPin152.AppScalingMultiplier :=1;
boPin152.AppScalingOffset :=0;
boPin152.AppUnit :="";
boPin152.CanDefault :=0;
boPin152.CanInit :=0;
boPin152.CanMax :=1;
boPin152.CanMin :=0;
boPin152.CanUnit :="";
boPin152.Description :="for the Neotec diag pages";
boPin152.ErrorReaction := eErrorReaction.ERSIG_DFLT;
boPin152.ReceiverAdress :=1;
boPin152.ToolScalingDivisor :=1;
boPin152.ToolScalingMultiplier :=1;
boPin152.ToolScalingOffset :=0;
boPin152.ToolUnit :="";

boPin176.AppScalingDivisor :=1;
boPin176.AppScalingMultiplier :=1;
boPin176.AppScalingOffset :=0;
boPin176.AppUnit :="";
boPin176.CanDefault :=0;
boPin176.CanInit :=0;
boPin176.CanMax :=1;
boPin176.CanMin :=0;
boPin176.CanUnit :="";
boPin176.Description :="for the Neotec diag pages";
boPin176.ErrorReaction := eErrorReaction.ERSIG_DFLT;
boPin176.ReceiverAdress :=1;
boPin176.ToolScalingDivisor :=1;
boPin176.ToolScalingMultiplier :=1;
boPin176.ToolScalingOffset :=0;
boPin176.ToolUnit :="";

boPin155.AppScalingDivisor :=1;
boPin155.AppScalingMultiplier :=1;
boPin155.AppScalingOffset :=0;
boPin155.AppUnit :="";
boPin155.CanDefault :=0;
boPin155.CanInit :=0;
boPin155.CanMax :=1;
boPin155.CanMin :=0;
boPin155.CanUnit :="";
boPin155.Description :="for the Neotec diag pages";
boPin155.ErrorReaction := eErrorReaction.ERSIG_DFLT;
boPin155.ReceiverAdress :=1;
boPin155.ToolScalingDivisor :=1;
boPin155.ToolScalingMultiplier :=1;
boPin155.ToolScalingOffset :=0;
boPin155.ToolUnit :="";

boPin179.AppScalingDivisor :=1;
boPin179.AppScalingMultiplier :=1;
boPin179.AppScalingOffset :=0;
boPin179.AppUnit :="";
boPin179.CanDefault :=0;
boPin179.CanInit :=0;
boPin179.CanMax :=1;
boPin179.CanMin :=0;
boPin179.CanUnit :="";
boPin179.Description :="for the Neotec diag pages";
boPin179.ErrorReaction := eErrorReaction.ERSIG_DFLT;
boPin179.ReceiverAdress :=1;
boPin179.ToolScalingDivisor :=1;
boPin179.ToolScalingMultiplier :=1;
boPin179.ToolScalingOffset :=0;
boPin179.ToolUnit :="";

boPin158.AppScalingDivisor :=1;
boPin158.AppScalingMultiplier :=1;
boPin158.AppScalingOffset :=0;
boPin158.AppUnit :="";
boPin158.CanDefault :=0;
boPin158.CanInit :=0;
boPin158.CanMax :=1;
boPin158.CanMin :=0;
boPin158.CanUnit :="";
boPin158.Description :="for the Neotec diag pages";
boPin158.ErrorReaction := eErrorReaction.ERSIG_DFLT;
boPin158.ReceiverAdress :=1;
boPin158.ToolScalingDivisor :=1;
boPin158.ToolScalingMultiplier :=1;
boPin158.ToolScalingOffset :=0;
boPin158.ToolUnit :="";

boPin182.AppScalingDivisor :=1;
boPin182.AppScalingMultiplier :=1;
boPin182.AppScalingOffset :=0;
boPin182.AppUnit :="";
boPin182.CanDefault :=0;
boPin182.CanInit :=0;
boPin182.CanMax :=1;
boPin182.CanMin :=0;
boPin182.CanUnit :="";
boPin182.Description :="for the Neotec diag pages";
boPin182.ErrorReaction := eErrorReaction.ERSIG_DFLT;
boPin182.ReceiverAdress :=1;
boPin182.ToolScalingDivisor :=1;
boPin182.ToolScalingMultiplier :=1;
boPin182.ToolScalingOffset :=0;
boPin182.ToolUnit :="";

boPin252.AppScalingDivisor :=1;
boPin252.AppScalingMultiplier :=1;
boPin252.AppScalingOffset :=0;
boPin252.AppUnit :="";
boPin252.CanDefault :=0;
boPin252.CanInit :=0;
boPin252.CanMax :=1;
boPin252.CanMin :=0;
boPin252.CanUnit :="";
boPin252.Description :="for the Neotec diag pages";
boPin252.ErrorReaction := eErrorReaction.ERSIG_DFLT;
boPin252.ReceiverAdress :=1;
boPin252.ToolScalingDivisor :=1;
boPin252.ToolScalingMultiplier :=1;
boPin252.ToolScalingOffset :=0;
boPin252.ToolUnit :="";

boPin239.AppScalingDivisor :=1;
boPin239.AppScalingMultiplier :=1;
boPin239.AppScalingOffset :=0;
boPin239.AppUnit :="";
boPin239.CanDefault :=0;
boPin239.CanInit :=0;
boPin239.CanMax :=1;
boPin239.CanMin :=0;
boPin239.CanUnit :="";
boPin239.Description :="for the Neotec diag pages";
boPin239.ErrorReaction := eErrorReaction.ERSIG_DFLT;
boPin239.ReceiverAdress :=1;
boPin239.ToolScalingDivisor :=1;
boPin239.ToolScalingMultiplier :=1;
boPin239.ToolScalingOffset :=0;
boPin239.ToolUnit :="";

boPin188.AppScalingDivisor :=1;
boPin188.AppScalingMultiplier :=1;
boPin188.AppScalingOffset :=0;
boPin188.AppUnit :="";
boPin188.CanDefault :=0;
boPin188.CanInit :=0;
boPin188.CanMax :=1;
boPin188.CanMin :=0;
boPin188.CanUnit :="";
boPin188.Description :="for the Neotec diag pages";
boPin188.ErrorReaction := eErrorReaction.ERSIG_DFLT;
boPin188.ReceiverAdress :=1;
boPin188.ToolScalingDivisor :=1;
boPin188.ToolScalingMultiplier :=1;
boPin188.ToolScalingOffset :=0;
boPin188.ToolUnit :="";

boPin164.AppScalingDivisor :=1;
boPin164.AppScalingMultiplier :=1;
boPin164.AppScalingOffset :=0;
boPin164.AppUnit :="";
boPin164.CanDefault :=0;
boPin164.CanInit :=0;
boPin164.CanMax :=1;
boPin164.CanMin :=0;
boPin164.CanUnit :="";
boPin164.Description :="for the Neotec diag pages";
boPin164.ErrorReaction := eErrorReaction.ERSIG_DFLT;
boPin164.ReceiverAdress :=1;
boPin164.ToolScalingDivisor :=1;
boPin164.ToolScalingMultiplier :=1;
boPin164.ToolScalingOffset :=0;
boPin164.ToolUnit :="";

boPin191.AppScalingDivisor :=1;
boPin191.AppScalingMultiplier :=1;
boPin191.AppScalingOffset :=0;
boPin191.AppUnit :="";
boPin191.CanDefault :=0;
boPin191.CanInit :=0;
boPin191.CanMax :=1;
boPin191.CanMin :=0;
boPin191.CanUnit :="";
boPin191.Description :="for the Neotec diag pages";
boPin191.ErrorReaction := eErrorReaction.ERSIG_DFLT;
boPin191.ReceiverAdress :=1;
boPin191.ToolScalingDivisor :=1;
boPin191.ToolScalingMultiplier :=1;
boPin191.ToolScalingOffset :=0;
boPin191.ToolUnit :="";

boPin167.AppScalingDivisor :=1;
boPin167.AppScalingMultiplier :=1;
boPin167.AppScalingOffset :=0;
boPin167.AppUnit :="";
boPin167.CanDefault :=0;
boPin167.CanInit :=0;
boPin167.CanMax :=1;
boPin167.CanMin :=0;
boPin167.CanUnit :="";
boPin167.Description :="for the Neotec diag pages";
boPin167.ErrorReaction := eErrorReaction.ERSIG_DFLT;
boPin167.ReceiverAdress :=1;
boPin167.ToolScalingDivisor :=1;
boPin167.ToolScalingMultiplier :=1;
boPin167.ToolScalingOffset :=0;
boPin167.ToolUnit :="";

boPin194.AppScalingDivisor :=1;
boPin194.AppScalingMultiplier :=1;
boPin194.AppScalingOffset :=0;
boPin194.AppUnit :="";
boPin194.CanDefault :=0;
boPin194.CanInit :=0;
boPin194.CanMax :=1;
boPin194.CanMin :=0;
boPin194.CanUnit :="";
boPin194.Description :="for the Neotec diag pages";
boPin194.ErrorReaction := eErrorReaction.ERSIG_DFLT;
boPin194.ReceiverAdress :=1;
boPin194.ToolScalingDivisor :=1;
boPin194.ToolScalingMultiplier :=1;
boPin194.ToolScalingOffset :=0;
boPin194.ToolUnit :="";

boPin170.AppScalingDivisor :=1;
boPin170.AppScalingMultiplier :=1;
boPin170.AppScalingOffset :=0;
boPin170.AppUnit :="";
boPin170.CanDefault :=0;
boPin170.CanInit :=0;
boPin170.CanMax :=1;
boPin170.CanMin :=0;
boPin170.CanUnit :="";
boPin170.Description :="for the Neotec diag pages";
boPin170.ErrorReaction := eErrorReaction.ERSIG_DFLT;
boPin170.ReceiverAdress :=1;
boPin170.ToolScalingDivisor :=1;
boPin170.ToolScalingMultiplier :=1;
boPin170.ToolScalingOffset :=0;
boPin170.ToolUnit :="";

boPin192.AppScalingDivisor :=1;
boPin192.AppScalingMultiplier :=1;
boPin192.AppScalingOffset :=0;
boPin192.AppUnit :="";
boPin192.CanDefault :=0;
boPin192.CanInit :=0;
boPin192.CanMax :=1;
boPin192.CanMin :=0;
boPin192.CanUnit :="";
boPin192.Description :="for the Neotec diag pages";
boPin192.ErrorReaction := eErrorReaction.ERSIG_DFLT;
boPin192.ReceiverAdress :=1;
boPin192.ToolScalingDivisor :=1;
boPin192.ToolScalingMultiplier :=1;
boPin192.ToolScalingOffset :=0;
boPin192.ToolUnit :="";

boPin168.AppScalingDivisor :=1;
boPin168.AppScalingMultiplier :=1;
boPin168.AppScalingOffset :=0;
boPin168.AppUnit :="";
boPin168.CanDefault :=0;
boPin168.CanInit :=0;
boPin168.CanMax :=1;
boPin168.CanMin :=0;
boPin168.CanUnit :="";
boPin168.Description :="for the Neotec diag pages";
boPin168.ErrorReaction := eErrorReaction.ERSIG_DFLT;
boPin168.ReceiverAdress :=1;
boPin168.ToolScalingDivisor :=1;
boPin168.ToolScalingMultiplier :=1;
boPin168.ToolScalingOffset :=0;
boPin168.ToolUnit :="";


                
END_METHOD
END_FUNCTION_BLOCK

FUNCTION_BLOCK Msg8C0SendToEvision7MessageClass EXTENDS CanReceiveMessageClass
  VAR_INPUT
    boPin136_48XSFault : BoolCanSignalClass;
    boPin148_48XSFault : BoolCanSignalClass;
    boPin135_48XSFault : BoolCanSignalClass;
    boPin147_48XSFault : BoolCanSignalClass;
    boPin269_48XSFault : BoolCanSignalClass;
    boPin118_48XSFault : BoolCanSignalClass;
    boPin106_48XSFault : BoolCanSignalClass;
    boPin117_48XSFault : BoolCanSignalClass;
    boPin105_48XSFault : BoolCanSignalClass;
    boPin116_48XSFault : BoolCanSignalClass;
    boPin104_48XSFault : BoolCanSignalClass;
    boPin115_48XSFault : BoolCanSignalClass;
    boPin103_48XSFault : BoolCanSignalClass;
    boPin120_48XSFault : BoolCanSignalClass;
    boPin108_48XSFault : BoolCanSignalClass;
    boPin119_48XSFault : BoolCanSignalClass;
    boPin107_48XSFault : BoolCanSignalClass;
    boPin144_48XSFault : BoolCanSignalClass;
    boPin132_48XSFault : BoolCanSignalClass;
    boPin143_48XSFault : BoolCanSignalClass;
    boPin131_48XSFault : BoolCanSignalClass;
    boPin142_48XSFault : BoolCanSignalClass;
    boPin130_48XSFault : BoolCanSignalClass;
    boPin141_48XSFault : BoolCanSignalClass;
    boPin129_48XSFault : BoolCanSignalClass;
    boPin152_48XSFault : BoolCanSignalClass;
    boPin140_48XSFault : BoolCanSignalClass;
    boPin151_48XSFault : BoolCanSignalClass;
    boPin139_48XSFault : BoolCanSignalClass;
    boPin150_48XSFault : BoolCanSignalClass;
    boPin138_48XSFault : BoolCanSignalClass;
    boPin149_48XSFault : BoolCanSignalClass;
    boPin137_48XSFault : BoolCanSignalClass;
    boPin126_48XSFault : BoolCanSignalClass;
    boPin114_48XSFault : BoolCanSignalClass;
    boPin125_48XSFault : BoolCanSignalClass;
    boPin113_48XSFault : BoolCanSignalClass;
    boPin124_48XSFault : BoolCanSignalClass;
    boPin112_48XSFault : BoolCanSignalClass;
    boPin123_48XSFault : BoolCanSignalClass;
    boPin111_48XSFault : BoolCanSignalClass;
    boPin133_48XSFault : BoolCanSignalClass;
    boPin134_48XSFault : BoolCanSignalClass;
    boPin145_48XSFault : BoolCanSignalClass;
    boPin146_48XSFault : BoolCanSignalClass;
    boPin263_48XSFault : BoolCanSignalClass;
    boPin256_48XSFault : BoolCanSignalClass;
    boPin262_48XSFault : BoolCanSignalClass;
    boPin255_48XSFault : BoolCanSignalClass;
    boPin261_48XSFault : BoolCanSignalClass;
    boPin254_48XSFault : BoolCanSignalClass;
    boPin260_48XSFault : BoolCanSignalClass;
    boPin253_48XSFault : BoolCanSignalClass;
    boPin270_48XSFault : BoolCanSignalClass;
    boPin276_48XSFault : BoolCanSignalClass;
    boPin277_48XSFault : BoolCanSignalClass;
    boPin275_48XSFault : BoolCanSignalClass;
    boPin268_48XSFault : BoolCanSignalClass;
    boPin274_48XSFault : BoolCanSignalClass;
    boPin267_48XSFault : BoolCanSignalClass;
    Counter : UInt32CanSignalClass;
  END_VAR

            
          

METHOD SetData
  VAR_INPUT
    CanMsgPointer : POINTER TO CanMessageClass;
  END_VAR
                  IF IsValidPointer(canMsgPointer,'SetData') THEN
	SUPER^.SetData(CanMsgPointer);
	//Set the new data
	boPin136_48XSFault.Value := canMsgPointer^.GetBoolOnBit(0);
	boPin148_48XSFault.Value := canMsgPointer^.GetBoolOnBit(1);
	boPin135_48XSFault.Value := canMsgPointer^.GetBoolOnBit(2);
	boPin147_48XSFault.Value := canMsgPointer^.GetBoolOnBit(3);
	boPin269_48XSFault.Value := canMsgPointer^.GetBoolOnBit(4);
	boPin118_48XSFault.Value := canMsgPointer^.GetBoolOnBit(5);
	boPin106_48XSFault.Value := canMsgPointer^.GetBoolOnBit(6);
	boPin117_48XSFault.Value := canMsgPointer^.GetBoolOnBit(7);
	boPin105_48XSFault.Value := canMsgPointer^.GetBoolOnBit(8);
	boPin116_48XSFault.Value := canMsgPointer^.GetBoolOnBit(9);
	boPin104_48XSFault.Value := canMsgPointer^.GetBoolOnBit(10);
	boPin115_48XSFault.Value := canMsgPointer^.GetBoolOnBit(11);
	boPin103_48XSFault.Value := canMsgPointer^.GetBoolOnBit(12);
	boPin120_48XSFault.Value := canMsgPointer^.GetBoolOnBit(13);
	boPin108_48XSFault.Value := canMsgPointer^.GetBoolOnBit(14);
	boPin119_48XSFault.Value := canMsgPointer^.GetBoolOnBit(15);
	boPin107_48XSFault.Value := canMsgPointer^.GetBoolOnBit(16);
	boPin144_48XSFault.Value := canMsgPointer^.GetBoolOnBit(17);
	boPin132_48XSFault.Value := canMsgPointer^.GetBoolOnBit(18);
	boPin143_48XSFault.Value := canMsgPointer^.GetBoolOnBit(19);
	boPin131_48XSFault.Value := canMsgPointer^.GetBoolOnBit(20);
	boPin142_48XSFault.Value := canMsgPointer^.GetBoolOnBit(21);
	boPin130_48XSFault.Value := canMsgPointer^.GetBoolOnBit(22);
	boPin141_48XSFault.Value := canMsgPointer^.GetBoolOnBit(23);
	boPin129_48XSFault.Value := canMsgPointer^.GetBoolOnBit(24);
	boPin152_48XSFault.Value := canMsgPointer^.GetBoolOnBit(25);
	boPin140_48XSFault.Value := canMsgPointer^.GetBoolOnBit(26);
	boPin151_48XSFault.Value := canMsgPointer^.GetBoolOnBit(27);
	boPin139_48XSFault.Value := canMsgPointer^.GetBoolOnBit(28);
	boPin150_48XSFault.Value := canMsgPointer^.GetBoolOnBit(29);
	boPin138_48XSFault.Value := canMsgPointer^.GetBoolOnBit(30);
	boPin149_48XSFault.Value := canMsgPointer^.GetBoolOnBit(31);
	boPin137_48XSFault.Value := canMsgPointer^.GetBoolOnBit(32);
	boPin126_48XSFault.Value := canMsgPointer^.GetBoolOnBit(33);
	boPin114_48XSFault.Value := canMsgPointer^.GetBoolOnBit(34);
	boPin125_48XSFault.Value := canMsgPointer^.GetBoolOnBit(35);
	boPin113_48XSFault.Value := canMsgPointer^.GetBoolOnBit(36);
	boPin124_48XSFault.Value := canMsgPointer^.GetBoolOnBit(37);
	boPin112_48XSFault.Value := canMsgPointer^.GetBoolOnBit(38);
	boPin123_48XSFault.Value := canMsgPointer^.GetBoolOnBit(39);
	boPin111_48XSFault.Value := canMsgPointer^.GetBoolOnBit(40);
	boPin133_48XSFault.Value := canMsgPointer^.GetBoolOnBit(41);
	boPin134_48XSFault.Value := canMsgPointer^.GetBoolOnBit(42);
	boPin145_48XSFault.Value := canMsgPointer^.GetBoolOnBit(43);
	boPin146_48XSFault.Value := canMsgPointer^.GetBoolOnBit(44);
	boPin263_48XSFault.Value := canMsgPointer^.GetBoolOnBit(45);
	boPin256_48XSFault.Value := canMsgPointer^.GetBoolOnBit(46);
	boPin262_48XSFault.Value := canMsgPointer^.GetBoolOnBit(47);
	boPin255_48XSFault.Value := canMsgPointer^.GetBoolOnBit(48);
	boPin261_48XSFault.Value := canMsgPointer^.GetBoolOnBit(49);
	boPin254_48XSFault.Value := canMsgPointer^.GetBoolOnBit(50);
	boPin260_48XSFault.Value := canMsgPointer^.GetBoolOnBit(51);
	boPin253_48XSFault.Value := canMsgPointer^.GetBoolOnBit(52);
	boPin270_48XSFault.Value := canMsgPointer^.GetBoolOnBit(53);
	boPin276_48XSFault.Value := canMsgPointer^.GetBoolOnBit(54);
	boPin277_48XSFault.Value := canMsgPointer^.GetBoolOnBit(55);
	boPin275_48XSFault.Value := canMsgPointer^.GetBoolOnBit(56);
	boPin268_48XSFault.Value := canMsgPointer^.GetBoolOnBit(57);
	boPin274_48XSFault.Value := canMsgPointer^.GetBoolOnBit(58);
	boPin267_48XSFault.Value := canMsgPointer^.GetBoolOnBit(59);
	//And increase the counter
	Counter.Value := CanMsgPointer^.Counter.Value;
END_IF

                
END_METHOD

PROPERTY boPin136_48XSFaultRawValue : BOOL
GET
                    boPin136_48XSFaultRawValue := boPin136_48XSFault.Value;

                  
END_GET
END_PROPERTY

PROPERTY boPin148_48XSFaultRawValue : BOOL
GET
                    boPin148_48XSFaultRawValue := boPin148_48XSFault.Value;

                  
END_GET
END_PROPERTY

PROPERTY boPin135_48XSFaultRawValue : BOOL
GET
                    boPin135_48XSFaultRawValue := boPin135_48XSFault.Value;

                  
END_GET
END_PROPERTY

PROPERTY boPin147_48XSFaultRawValue : BOOL
GET
                    boPin147_48XSFaultRawValue := boPin147_48XSFault.Value;

                  
END_GET
END_PROPERTY

PROPERTY boPin269_48XSFaultRawValue : BOOL
GET
                    boPin269_48XSFaultRawValue := boPin269_48XSFault.Value;

                  
END_GET
END_PROPERTY

PROPERTY boPin118_48XSFaultRawValue : BOOL
GET
                    boPin118_48XSFaultRawValue := boPin118_48XSFault.Value;

                  
END_GET
END_PROPERTY

PROPERTY boPin106_48XSFaultRawValue : BOOL
GET
                    boPin106_48XSFaultRawValue := boPin106_48XSFault.Value;

                  
END_GET
END_PROPERTY

PROPERTY boPin117_48XSFaultRawValue : BOOL
GET
                    boPin117_48XSFaultRawValue := boPin117_48XSFault.Value;

                  
END_GET
END_PROPERTY

PROPERTY boPin105_48XSFaultRawValue : BOOL
GET
                    boPin105_48XSFaultRawValue := boPin105_48XSFault.Value;

                  
END_GET
END_PROPERTY

PROPERTY boPin116_48XSFaultRawValue : BOOL
GET
                    boPin116_48XSFaultRawValue := boPin116_48XSFault.Value;

                  
END_GET
END_PROPERTY

PROPERTY boPin104_48XSFaultRawValue : BOOL
GET
                    boPin104_48XSFaultRawValue := boPin104_48XSFault.Value;

                  
END_GET
END_PROPERTY

PROPERTY boPin115_48XSFaultRawValue : BOOL
GET
                    boPin115_48XSFaultRawValue := boPin115_48XSFault.Value;

                  
END_GET
END_PROPERTY

PROPERTY boPin103_48XSFaultRawValue : BOOL
GET
                    boPin103_48XSFaultRawValue := boPin103_48XSFault.Value;

                  
END_GET
END_PROPERTY

PROPERTY boPin120_48XSFaultRawValue : BOOL
GET
                    boPin120_48XSFaultRawValue := boPin120_48XSFault.Value;

                  
END_GET
END_PROPERTY

PROPERTY boPin108_48XSFaultRawValue : BOOL
GET
                    boPin108_48XSFaultRawValue := boPin108_48XSFault.Value;

                  
END_GET
END_PROPERTY

PROPERTY boPin119_48XSFaultRawValue : BOOL
GET
                    boPin119_48XSFaultRawValue := boPin119_48XSFault.Value;

                  
END_GET
END_PROPERTY

PROPERTY boPin107_48XSFaultRawValue : BOOL
GET
                    boPin107_48XSFaultRawValue := boPin107_48XSFault.Value;

                  
END_GET
END_PROPERTY

PROPERTY boPin144_48XSFaultRawValue : BOOL
GET
                    boPin144_48XSFaultRawValue := boPin144_48XSFault.Value;

                  
END_GET
END_PROPERTY

PROPERTY boPin132_48XSFaultRawValue : BOOL
GET
                    boPin132_48XSFaultRawValue := boPin132_48XSFault.Value;

                  
END_GET
END_PROPERTY

PROPERTY boPin143_48XSFaultRawValue : BOOL
GET
                    boPin143_48XSFaultRawValue := boPin143_48XSFault.Value;

                  
END_GET
END_PROPERTY

PROPERTY boPin131_48XSFaultRawValue : BOOL
GET
                    boPin131_48XSFaultRawValue := boPin131_48XSFault.Value;

                  
END_GET
END_PROPERTY

PROPERTY boPin142_48XSFaultRawValue : BOOL
GET
                    boPin142_48XSFaultRawValue := boPin142_48XSFault.Value;

                  
END_GET
END_PROPERTY

PROPERTY boPin130_48XSFaultRawValue : BOOL
GET
                    boPin130_48XSFaultRawValue := boPin130_48XSFault.Value;

                  
END_GET
END_PROPERTY

PROPERTY boPin141_48XSFaultRawValue : BOOL
GET
                    boPin141_48XSFaultRawValue := boPin141_48XSFault.Value;

                  
END_GET
END_PROPERTY

PROPERTY boPin129_48XSFaultRawValue : BOOL
GET
                    boPin129_48XSFaultRawValue := boPin129_48XSFault.Value;

                  
END_GET
END_PROPERTY

PROPERTY boPin152_48XSFaultRawValue : BOOL
GET
                    boPin152_48XSFaultRawValue := boPin152_48XSFault.Value;

                  
END_GET
END_PROPERTY

PROPERTY boPin140_48XSFaultRawValue : BOOL
GET
                    boPin140_48XSFaultRawValue := boPin140_48XSFault.Value;

                  
END_GET
END_PROPERTY

PROPERTY boPin151_48XSFaultRawValue : BOOL
GET
                    boPin151_48XSFaultRawValue := boPin151_48XSFault.Value;

                  
END_GET
END_PROPERTY

PROPERTY boPin139_48XSFaultRawValue : BOOL
GET
                    boPin139_48XSFaultRawValue := boPin139_48XSFault.Value;

                  
END_GET
END_PROPERTY

PROPERTY boPin150_48XSFaultRawValue : BOOL
GET
                    boPin150_48XSFaultRawValue := boPin150_48XSFault.Value;

                  
END_GET
END_PROPERTY

PROPERTY boPin138_48XSFaultRawValue : BOOL
GET
                    boPin138_48XSFaultRawValue := boPin138_48XSFault.Value;

                  
END_GET
END_PROPERTY

PROPERTY boPin149_48XSFaultRawValue : BOOL
GET
                    boPin149_48XSFaultRawValue := boPin149_48XSFault.Value;

                  
END_GET
END_PROPERTY

PROPERTY boPin137_48XSFaultRawValue : BOOL
GET
                    boPin137_48XSFaultRawValue := boPin137_48XSFault.Value;

                  
END_GET
END_PROPERTY

PROPERTY boPin126_48XSFaultRawValue : BOOL
GET
                    boPin126_48XSFaultRawValue := boPin126_48XSFault.Value;

                  
END_GET
END_PROPERTY

PROPERTY boPin114_48XSFaultRawValue : BOOL
GET
                    boPin114_48XSFaultRawValue := boPin114_48XSFault.Value;

                  
END_GET
END_PROPERTY

PROPERTY boPin125_48XSFaultRawValue : BOOL
GET
                    boPin125_48XSFaultRawValue := boPin125_48XSFault.Value;

                  
END_GET
END_PROPERTY

PROPERTY boPin113_48XSFaultRawValue : BOOL
GET
                    boPin113_48XSFaultRawValue := boPin113_48XSFault.Value;

                  
END_GET
END_PROPERTY

PROPERTY boPin124_48XSFaultRawValue : BOOL
GET
                    boPin124_48XSFaultRawValue := boPin124_48XSFault.Value;

                  
END_GET
END_PROPERTY

PROPERTY boPin112_48XSFaultRawValue : BOOL
GET
                    boPin112_48XSFaultRawValue := boPin112_48XSFault.Value;

                  
END_GET
END_PROPERTY

PROPERTY boPin123_48XSFaultRawValue : BOOL
GET
                    boPin123_48XSFaultRawValue := boPin123_48XSFault.Value;

                  
END_GET
END_PROPERTY

PROPERTY boPin111_48XSFaultRawValue : BOOL
GET
                    boPin111_48XSFaultRawValue := boPin111_48XSFault.Value;

                  
END_GET
END_PROPERTY

PROPERTY boPin133_48XSFaultRawValue : BOOL
GET
                    boPin133_48XSFaultRawValue := boPin133_48XSFault.Value;

                  
END_GET
END_PROPERTY

PROPERTY boPin134_48XSFaultRawValue : BOOL
GET
                    boPin134_48XSFaultRawValue := boPin134_48XSFault.Value;

                  
END_GET
END_PROPERTY

PROPERTY boPin145_48XSFaultRawValue : BOOL
GET
                    boPin145_48XSFaultRawValue := boPin145_48XSFault.Value;

                  
END_GET
END_PROPERTY

PROPERTY boPin146_48XSFaultRawValue : BOOL
GET
                    boPin146_48XSFaultRawValue := boPin146_48XSFault.Value;

                  
END_GET
END_PROPERTY

PROPERTY boPin263_48XSFaultRawValue : BOOL
GET
                    boPin263_48XSFaultRawValue := boPin263_48XSFault.Value;

                  
END_GET
END_PROPERTY

PROPERTY boPin256_48XSFaultRawValue : BOOL
GET
                    boPin256_48XSFaultRawValue := boPin256_48XSFault.Value;

                  
END_GET
END_PROPERTY

PROPERTY boPin262_48XSFaultRawValue : BOOL
GET
                    boPin262_48XSFaultRawValue := boPin262_48XSFault.Value;

                  
END_GET
END_PROPERTY

PROPERTY boPin255_48XSFaultRawValue : BOOL
GET
                    boPin255_48XSFaultRawValue := boPin255_48XSFault.Value;

                  
END_GET
END_PROPERTY

PROPERTY boPin261_48XSFaultRawValue : BOOL
GET
                    boPin261_48XSFaultRawValue := boPin261_48XSFault.Value;

                  
END_GET
END_PROPERTY

PROPERTY boPin254_48XSFaultRawValue : BOOL
GET
                    boPin254_48XSFaultRawValue := boPin254_48XSFault.Value;

                  
END_GET
END_PROPERTY

PROPERTY boPin260_48XSFaultRawValue : BOOL
GET
                    boPin260_48XSFaultRawValue := boPin260_48XSFault.Value;

                  
END_GET
END_PROPERTY

PROPERTY boPin253_48XSFaultRawValue : BOOL
GET
                    boPin253_48XSFaultRawValue := boPin253_48XSFault.Value;

                  
END_GET
END_PROPERTY

PROPERTY boPin270_48XSFaultRawValue : BOOL
GET
                    boPin270_48XSFaultRawValue := boPin270_48XSFault.Value;

                  
END_GET
END_PROPERTY

PROPERTY boPin276_48XSFaultRawValue : BOOL
GET
                    boPin276_48XSFaultRawValue := boPin276_48XSFault.Value;

                  
END_GET
END_PROPERTY

PROPERTY boPin277_48XSFaultRawValue : BOOL
GET
                    boPin277_48XSFaultRawValue := boPin277_48XSFault.Value;

                  
END_GET
END_PROPERTY

PROPERTY boPin275_48XSFaultRawValue : BOOL
GET
                    boPin275_48XSFaultRawValue := boPin275_48XSFault.Value;

                  
END_GET
END_PROPERTY

PROPERTY boPin268_48XSFaultRawValue : BOOL
GET
                    boPin268_48XSFaultRawValue := boPin268_48XSFault.Value;

                  
END_GET
END_PROPERTY

PROPERTY boPin274_48XSFaultRawValue : BOOL
GET
                    boPin274_48XSFaultRawValue := boPin274_48XSFault.Value;

                  
END_GET
END_PROPERTY

PROPERTY boPin267_48XSFaultRawValue : BOOL
GET
                    boPin267_48XSFaultRawValue := boPin267_48XSFault.Value;

                  
END_GET
END_PROPERTY

PROPERTY boPin136_48XSFaultToolValue : BOOL
GET
                    boPin136_48XSFaultToolValue := boPin136_48XSFault.Value;

                  
END_GET
END_PROPERTY

PROPERTY boPin148_48XSFaultToolValue : BOOL
GET
                    boPin148_48XSFaultToolValue := boPin148_48XSFault.Value;

                  
END_GET
END_PROPERTY

PROPERTY boPin135_48XSFaultToolValue : BOOL
GET
                    boPin135_48XSFaultToolValue := boPin135_48XSFault.Value;

                  
END_GET
END_PROPERTY

PROPERTY boPin147_48XSFaultToolValue : BOOL
GET
                    boPin147_48XSFaultToolValue := boPin147_48XSFault.Value;

                  
END_GET
END_PROPERTY

PROPERTY boPin269_48XSFaultToolValue : BOOL
GET
                    boPin269_48XSFaultToolValue := boPin269_48XSFault.Value;

                  
END_GET
END_PROPERTY

PROPERTY boPin118_48XSFaultToolValue : BOOL
GET
                    boPin118_48XSFaultToolValue := boPin118_48XSFault.Value;

                  
END_GET
END_PROPERTY

PROPERTY boPin106_48XSFaultToolValue : BOOL
GET
                    boPin106_48XSFaultToolValue := boPin106_48XSFault.Value;

                  
END_GET
END_PROPERTY

PROPERTY boPin117_48XSFaultToolValue : BOOL
GET
                    boPin117_48XSFaultToolValue := boPin117_48XSFault.Value;

                  
END_GET
END_PROPERTY

PROPERTY boPin105_48XSFaultToolValue : BOOL
GET
                    boPin105_48XSFaultToolValue := boPin105_48XSFault.Value;

                  
END_GET
END_PROPERTY

PROPERTY boPin116_48XSFaultToolValue : BOOL
GET
                    boPin116_48XSFaultToolValue := boPin116_48XSFault.Value;

                  
END_GET
END_PROPERTY

PROPERTY boPin104_48XSFaultToolValue : BOOL
GET
                    boPin104_48XSFaultToolValue := boPin104_48XSFault.Value;

                  
END_GET
END_PROPERTY

PROPERTY boPin115_48XSFaultToolValue : BOOL
GET
                    boPin115_48XSFaultToolValue := boPin115_48XSFault.Value;

                  
END_GET
END_PROPERTY

PROPERTY boPin103_48XSFaultToolValue : BOOL
GET
                    boPin103_48XSFaultToolValue := boPin103_48XSFault.Value;

                  
END_GET
END_PROPERTY

PROPERTY boPin120_48XSFaultToolValue : BOOL
GET
                    boPin120_48XSFaultToolValue := boPin120_48XSFault.Value;

                  
END_GET
END_PROPERTY

PROPERTY boPin108_48XSFaultToolValue : BOOL
GET
                    boPin108_48XSFaultToolValue := boPin108_48XSFault.Value;

                  
END_GET
END_PROPERTY

PROPERTY boPin119_48XSFaultToolValue : BOOL
GET
                    boPin119_48XSFaultToolValue := boPin119_48XSFault.Value;

                  
END_GET
END_PROPERTY

PROPERTY boPin107_48XSFaultToolValue : BOOL
GET
                    boPin107_48XSFaultToolValue := boPin107_48XSFault.Value;

                  
END_GET
END_PROPERTY

PROPERTY boPin144_48XSFaultToolValue : BOOL
GET
                    boPin144_48XSFaultToolValue := boPin144_48XSFault.Value;

                  
END_GET
END_PROPERTY

PROPERTY boPin132_48XSFaultToolValue : BOOL
GET
                    boPin132_48XSFaultToolValue := boPin132_48XSFault.Value;

                  
END_GET
END_PROPERTY

PROPERTY boPin143_48XSFaultToolValue : BOOL
GET
                    boPin143_48XSFaultToolValue := boPin143_48XSFault.Value;

                  
END_GET
END_PROPERTY

PROPERTY boPin131_48XSFaultToolValue : BOOL
GET
                    boPin131_48XSFaultToolValue := boPin131_48XSFault.Value;

                  
END_GET
END_PROPERTY

PROPERTY boPin142_48XSFaultToolValue : BOOL
GET
                    boPin142_48XSFaultToolValue := boPin142_48XSFault.Value;

                  
END_GET
END_PROPERTY

PROPERTY boPin130_48XSFaultToolValue : BOOL
GET
                    boPin130_48XSFaultToolValue := boPin130_48XSFault.Value;

                  
END_GET
END_PROPERTY

PROPERTY boPin141_48XSFaultToolValue : BOOL
GET
                    boPin141_48XSFaultToolValue := boPin141_48XSFault.Value;

                  
END_GET
END_PROPERTY

PROPERTY boPin129_48XSFaultToolValue : BOOL
GET
                    boPin129_48XSFaultToolValue := boPin129_48XSFault.Value;

                  
END_GET
END_PROPERTY

PROPERTY boPin152_48XSFaultToolValue : BOOL
GET
                    boPin152_48XSFaultToolValue := boPin152_48XSFault.Value;

                  
END_GET
END_PROPERTY

PROPERTY boPin140_48XSFaultToolValue : BOOL
GET
                    boPin140_48XSFaultToolValue := boPin140_48XSFault.Value;

                  
END_GET
END_PROPERTY

PROPERTY boPin151_48XSFaultToolValue : BOOL
GET
                    boPin151_48XSFaultToolValue := boPin151_48XSFault.Value;

                  
END_GET
END_PROPERTY

PROPERTY boPin139_48XSFaultToolValue : BOOL
GET
                    boPin139_48XSFaultToolValue := boPin139_48XSFault.Value;

                  
END_GET
END_PROPERTY

PROPERTY boPin150_48XSFaultToolValue : BOOL
GET
                    boPin150_48XSFaultToolValue := boPin150_48XSFault.Value;

                  
END_GET
END_PROPERTY

PROPERTY boPin138_48XSFaultToolValue : BOOL
GET
                    boPin138_48XSFaultToolValue := boPin138_48XSFault.Value;

                  
END_GET
END_PROPERTY

PROPERTY boPin149_48XSFaultToolValue : BOOL
GET
                    boPin149_48XSFaultToolValue := boPin149_48XSFault.Value;

                  
END_GET
END_PROPERTY

PROPERTY boPin137_48XSFaultToolValue : BOOL
GET
                    boPin137_48XSFaultToolValue := boPin137_48XSFault.Value;

                  
END_GET
END_PROPERTY

PROPERTY boPin126_48XSFaultToolValue : BOOL
GET
                    boPin126_48XSFaultToolValue := boPin126_48XSFault.Value;

                  
END_GET
END_PROPERTY

PROPERTY boPin114_48XSFaultToolValue : BOOL
GET
                    boPin114_48XSFaultToolValue := boPin114_48XSFault.Value;

                  
END_GET
END_PROPERTY

PROPERTY boPin125_48XSFaultToolValue : BOOL
GET
                    boPin125_48XSFaultToolValue := boPin125_48XSFault.Value;

                  
END_GET
END_PROPERTY

PROPERTY boPin113_48XSFaultToolValue : BOOL
GET
                    boPin113_48XSFaultToolValue := boPin113_48XSFault.Value;

                  
END_GET
END_PROPERTY

PROPERTY boPin124_48XSFaultToolValue : BOOL
GET
                    boPin124_48XSFaultToolValue := boPin124_48XSFault.Value;

                  
END_GET
END_PROPERTY

PROPERTY boPin112_48XSFaultToolValue : BOOL
GET
                    boPin112_48XSFaultToolValue := boPin112_48XSFault.Value;

                  
END_GET
END_PROPERTY

PROPERTY boPin123_48XSFaultToolValue : BOOL
GET
                    boPin123_48XSFaultToolValue := boPin123_48XSFault.Value;

                  
END_GET
END_PROPERTY

PROPERTY boPin111_48XSFaultToolValue : BOOL
GET
                    boPin111_48XSFaultToolValue := boPin111_48XSFault.Value;

                  
END_GET
END_PROPERTY

PROPERTY boPin133_48XSFaultToolValue : BOOL
GET
                    boPin133_48XSFaultToolValue := boPin133_48XSFault.Value;

                  
END_GET
END_PROPERTY

PROPERTY boPin134_48XSFaultToolValue : BOOL
GET
                    boPin134_48XSFaultToolValue := boPin134_48XSFault.Value;

                  
END_GET
END_PROPERTY

PROPERTY boPin145_48XSFaultToolValue : BOOL
GET
                    boPin145_48XSFaultToolValue := boPin145_48XSFault.Value;

                  
END_GET
END_PROPERTY

PROPERTY boPin146_48XSFaultToolValue : BOOL
GET
                    boPin146_48XSFaultToolValue := boPin146_48XSFault.Value;

                  
END_GET
END_PROPERTY

PROPERTY boPin263_48XSFaultToolValue : BOOL
GET
                    boPin263_48XSFaultToolValue := boPin263_48XSFault.Value;

                  
END_GET
END_PROPERTY

PROPERTY boPin256_48XSFaultToolValue : BOOL
GET
                    boPin256_48XSFaultToolValue := boPin256_48XSFault.Value;

                  
END_GET
END_PROPERTY

PROPERTY boPin262_48XSFaultToolValue : BOOL
GET
                    boPin262_48XSFaultToolValue := boPin262_48XSFault.Value;

                  
END_GET
END_PROPERTY

PROPERTY boPin255_48XSFaultToolValue : BOOL
GET
                    boPin255_48XSFaultToolValue := boPin255_48XSFault.Value;

                  
END_GET
END_PROPERTY

